(* CoDeSys 2.3.9.47 project: Program-CHP-3.pro *)
(* Libraries: Util.lib 16.5.13 14:00:50, Standard.lib 20.5.14 08:13:26, Iecsfc.lib 16.5.13 14:00:50, SYSLIBCALLBACK.LIB 16.5.13 14:00:50, mod_com.lib 16.5.13 14:00:50, SerComm.lib 16.5.13 14:00:50, Serial_Interface_01.lib 22.4.13 12:50:14, Modb_l05.lib 13.5.15 10:30:08, SysLibTime.lib 16.5.13 14:00:48, SysLibFile.lib 16.5.13 14:00:50, SysLibDir.lib 16.5.13 14:00:50, SysLibMem.lib 16.5.13 14:00:50, WAGO_Datalogger_02.lib 21.4.17 00:23:22, SysLibSockets.lib 22.5.14 16:16:32, NETVARUDP_LIB_V23.LIB 14.6.13 10:36:42 *)

(* PLC configuration (modules and I/O channels)
xDI_24V_01 AT %IX86.0 [BOOLOnX_I] Ch_1 Digital input
xDI_24V_02 AT %IX86.1 [BOOLOnX_I] Ch_2 Digital input
xDI_24V_03 AT %IX86.2 [BOOLOnX_I] Ch_3 Digital input
xDI_24V_04 AT %IX86.3 [BOOLOnX_I] Ch_4 Digital input
xDI_24V_05 AT %IX86.4 [BOOLOnX_I] Ch_5 Digital input
xDI_24V_06 AT %IX86.5 [BOOLOnX_I] Ch_6 Digital input
xDI_24V_07 AT %IX86.6 [BOOLOnX_I] Ch_7 Digital input
xDI_24V_08 AT %IX86.7 [BOOLOnX_I] Ch_8 Digital input
xDO_24V_01 AT %QX24.0 [BOOLOnX_Q] Ch_1 Digital output
xDO_24V_02 AT %QX24.1 [BOOLOnX_Q] Ch_2 Digital output
xDO_24V_03 AT %QX24.2 [BOOLOnX_Q] Ch_3 Digital output
xDO_24V_04 AT %QX24.3 [BOOLOnX_Q] Ch_4 Digital output
xDO_24V_05 AT %QX24.4 [BOOLOnX_Q] Ch_5 Digital output
xDO_24V_06 AT %QX24.5 [BOOLOnX_Q] Ch_6 Digital output
xDO_24V_07 AT %QX24.6 [BOOLOnX_Q] Ch_7 Digital output
xDO_24V_08 AT %QX24.7 [BOOLOnX_Q] Ch_8 Digital output
xDO_24V_09 AT %QX24.8 [BOOLOnX_Q] Ch_1 Digital output
xDO_24V_10 AT %QX24.9 [BOOLOnX_Q] Ch_2 Digital output
xDO_24V_11 AT %QX24.10 [BOOLOnX_Q] Ch_3 Digital output
xDO_24V_12 AT %QX24.11 [BOOLOnX_Q] Ch_4 Digital output
xDO_24V_13 AT %QX24.12 [BOOLOnX_Q] Ch_5 Digital output
xDO_24V_14 AT %QX24.13 [BOOLOnX_Q] Ch_6 Digital output
xDO_24V_15 AT %QX24.14 [BOOLOnX_Q] Ch_7 Digital output
xDO_24V_16 AT %QX24.15 [BOOLOnX_Q] Ch_8 Digital output
AT %IB0 [BYTEOnB_I] First Byte of 24
AT %QB0 [BYTEOnB_Q] First Byte of 24
wAO_U_01 AT %QW12 [WORDOnW_Q] Ch_1 Analog output
wAO_U_02 AT %QW13 [WORDOnW_Q] Ch_2 Analog output
wAO_U_03 AT %QW14 [WORDOnW_Q] Ch_3 Analog output
wAO_U_04 AT %QW15 [WORDOnW_Q] Ch_4 Analog output
wAO_I_01 AT %QW16 [WORDOnW_Q] Ch_1 Analog output
wAO_I_02 AT %QW17 [WORDOnW_Q] Ch_2 Analog output
wAO_I_03 AT %QW18 [WORDOnW_Q] Ch_3 Analog output
wAO_I_04 AT %QW19 [WORDOnW_Q] Ch_4 Analog output
wAO_I_05 AT %QW20 [WORDOnW_Q] Ch_1 Analog output
wAO_I_06 AT %QW21 [WORDOnW_Q] Ch_2 Analog output
wAO_I_07 AT %QW22 [WORDOnW_Q] Ch_3 Analog output
wAO_I_08 AT %QW23 [WORDOnW_Q] Ch_4 Analog output
0750-0459 4 AI 0-10V DC s.e. [Type_8_4_Channels] node 7, in %IB188 out %QB88
  wAI_U_01 AT %IW12 [WORDOnW_I] Ch_1 Input word
  wAI_U_02 AT %IW13 [WORDOnW_I] Ch_2 Input word
  wAI_U_03 AT %IW14 [WORDOnW_I] Ch_3 Input word
  wAI_U_04 AT %IW15 [WORDOnW_I] Ch_4 Input word
0750-0455 4 AI 4-20mA s.e. [Type_8_4_Channels] node 8, in %IB188 out %QB96
  wAI_I_01 AT %IW16 [WORDOnW_I] Ch_1 Input word
  wAI_I_02 AT %IW17 [WORDOnW_I] Ch_2 Input word
  wAI_I_03 AT %IW18 [WORDOnW_I] Ch_3 Input word
  wAI_I_04 AT %IW19 [WORDOnW_I] Ch_4 Input word
  wAI_I_05 AT %IW20 [WORDOnW_I] Ch_1 Input word
  wAI_I_06 AT %IW21 [WORDOnW_I] Ch_2 Input word
  wAI_I_07 AT %IW22 [WORDOnW_I] Ch_3 Input word
  wAI_I_08 AT %IW23 [WORDOnW_I] Ch_4 Input word
0750-0469 2 AI Thermocouple / K / Diag. [Type_44_2_Channels] node 10, in %IB204 out %QB96
  iAI_PTTK_01 AT %IW24 [INTOnW_I] Ch_1 signed Input value
  iAI_PTTK_02 AT %IW25 [INTOnW_I] Ch_2 signed Input value
0750-0469 2 AI Thermocouple / K / Diag. [Type_44_2_Channels] node 11, in %IB212 out %QB96
  iAI_PTTK_03 AT %IW26 [INTOnW_I] Ch_1 signed Input value
  iAI_PTTK_04 AT %IW27 [INTOnW_I] Ch_2 signed Input value
0750-0469 2 AI Thermocouple / K / Diag. [Type_44_2_Channels] node 12, in %IB216 out %QB96
  iAI_PTTK_05 AT %IW28 [INTOnW_I] Ch_1 signed Input value
  iAI_PTTK_06 AT %IW29 [INTOnW_I] Ch_2 signed Input value
0750-0469 2 AI Thermocouple / K / Diag. [Type_44_2_Channels] node 13, in %IB220 out %QB96
  iAI_PTTK_07 AT %IW30 [INTOnW_I] Ch_1 signed Input value
  iAI_PTTK_08 AT %IW31 [INTOnW_I] Ch_2 signed Input value
0750-0469 2 AI Thermocouple / K / Diag. [Type_44_2_Channels] node 14, in %IB224 out %QB96
  iAI_PTTK_09 AT %IW32 [INTOnW_I] Ch_1 signed Input value
  iAI_PTTK_10 AT %IW33 [INTOnW_I] Ch_2 signed Input value
0750-0469 2 AI Thermocouple / K / Diag. [Type_44_2_Channels] node 15, in %IB228 out %QB96
  iAI_PTTK_11 AT %IW34 [INTOnW_I] Ch_1 signed Input value
  iAI_PTTK_12 AT %IW35 [INTOnW_I] Ch_2 signed Input value
0750-0469 2 AI Thermocouple / K / Diag. [Type_44_2_Channels] node 16, in %IB232 out %QB96
  iAI_PTTK_13 AT %IW36 [INTOnW_I] Ch_1 signed Input value
  iAI_PTTK_14 AT %IW37 [INTOnW_I] Ch_2 signed Input value
0750-0469 2 AI Thermocouple / K / Diag. [Type_44_2_Channels] node 17, in %IB236 out %QB96
  iAI_PTTK_15 AT %IW38 [INTOnW_I] Ch_1 signed Input value
  iAI_PTTK_16 AT %IW39 [INTOnW_I] Ch_2 signed Input value
0750-0469 2 AI Thermocouple / K / Diag. [Type_44_2_Channels] node 18, in %IB240 out %QB96
  iAI_PTTK_17 AT %IW40 [INTOnW_I] Ch_1 signed Input value
  iAI_PTTK_18 AT %IW41 [INTOnW_I] Ch_2 signed Input value
0750-0469 2 AI Thermocouple / K / Diag. [Type_44_2_Channels] node 19, in %IB244 out %QB96
  iAI_PTTK_19 AT %IW42 [INTOnW_I] Ch_1 signed Input value
  iAI_PTTK_20 AT %IW43 [INTOnW_I] Ch_2 signed Input value
0750-0469 2 AI Thermocouple / K / Diag. [Type_44_2_Channels] node 20, in %IB248 out %QB96
  iAI_PTTK_21 AT %IW44 [INTOnW_I] Ch_1 signed Input value
  iAI_PTTK_22 AT %IW45 [INTOnW_I] Ch_2 signed Input value
  iAI_PT100_01 AT %IW46 [INTOnW_I] Ch_1 signed Input value
  iAI_PT100_02 AT %IW47 [INTOnW_I] Ch_2 signed Input value
  iAI_PT100_03 AT %IW48 [INTOnW_I] Ch_1 signed Input value
  iAI_PT100_04 AT %IW49 [INTOnW_I] Ch_2 signed Input value
0750-0461 2 AI PT100 (RTD) [Type_44_2_Channels] node 23, in %IB260 out %QB96
  iAI_PT100_05 AT %IW50 [INTOnW_I] Ch_1 signed Input value
  iAI_PT100_06 AT %IW51 [INTOnW_I] Ch_2 signed Input value
0750-0461 2 AI PT100 (RTD) [Type_44_2_Channels] node 24, in %IB264 out %QB96
  iAI_PT100_07 AT %IW52 [INTOnW_I] Ch_1 signed Input value
  iAI_PT100_08 AT %IW53 [INTOnW_I] Ch_2 signed Input value
0750-0461 2 AI PT100 (RTD) [Type_44_2_Channels] node 25, in %IB268 out %QB96
  iAI_PT100_09 AT %IW54 [INTOnW_I] Ch_1 signed Input value
  iAI_PT100_10 AT %IW55 [INTOnW_I] Ch_2 signed Input value
0750-0461 2 AI PT100 (RTD) [Type_44_2_Channels] node 26, in %IB272 out %QB96
  iAI_PT100_11 AT %IW56 [INTOnW_I] Ch_1 signed Input value
  iAI_PT100_12 AT %IW57 [INTOnW_I] Ch_2 signed Input value
0750-0461 2 AI PT100 (RTD) [Type_44_2_Channels] node 27, in %IB276 out %QB96
  iAI_PT100_13 AT %IW58 [INTOnW_I] Ch_1 signed Input value
  iAI_PT100_14 AT %IW59 [INTOnW_I] Ch_2 signed Input value
0750-0461 2 AI PT100 (RTD) [Type_44_2_Channels] node 28, in %IB280 out %QB96
  iAI_PT100_15 AT %IW60 [INTOnW_I] Ch_1 signed Input value
  iAI_PT100_16 AT %IW61 [INTOnW_I] Ch_2 signed Input value
0750-0461 2 AI PT100 (RTD) [Type_44_2_Channels] node 29, in %IB284 out %QB96
  iAI_PT100_17 AT %IW62 [INTOnW_I] Ch_1 signed Input value
  iAI_PT100_18 AT %IW63 [INTOnW_I] Ch_2 signed Input value
0750-0461 2 AI PT100 (RTD) [Type_44_2_Channels] node 30, in %IB288 out %QB96
  iAI_PT100_19 AT %IW64 [INTOnW_I] Ch_1 signed Input value
  iAI_PT100_20 AT %IW65 [INTOnW_I] Ch_2 signed Input value
0750-0461 2 AI PT100 (RTD) [Type_44_2_Channels] node 31, in %IB292 out %QB96
  iAI_PT100_21 AT %IW66 [INTOnW_I] Ch_1 signed Input value
  iAI_PT100_22 AT %IW67 [INTOnW_I] Ch_2 signed Input value
0750-0461 2 AI PT100 (RTD) [Type_44_2_Channels] node 0, in %IB296 out %QB96
  iAI_PT100_23 AT %IW68 [INTOnW_I] Ch_1 signed Input value
  iAI_PT100_24 AT %IW69 [INTOnW_I] Ch_2 signed Input value
0750-0460 4 AI PT100 (RTD) [Type_44_4_Channels] node 32, in %IB300 out %QB96
  AT %IW70 [INTOnW_I] Ch_1 signed Input value
  AT %IW71 [INTOnW_I] Ch_2 signed Input value
  AT %IW72 [INTOnW_I] Ch_3 signed Input value
  AT %IW73 [INTOnW_I] Ch_4 signed Input value
0750-0460 4 AI PT100 (RTD) [Type_44_4_Channels] node 33, in %IB304 out %QB96
  AT %IW74 [INTOnW_I] Ch_1 signed Input value
  AT %IW75 [INTOnW_I] Ch_2 signed Input value
  AT %IW76 [INTOnW_I] Ch_3 signed Input value
  AT %IW77 [INTOnW_I] Ch_4 signed Input value
0750-0460 4 AI PT100 (RTD) [Type_44_4_Channels] node 34, in %IB312 out %QB96
  AT %IW78 [INTOnW_I] Ch_1 signed Input value
  AT %IW79 [INTOnW_I] Ch_2 signed Input value
  AT %IW80 [INTOnW_I] Ch_3 signed Input value
  AT %IW81 [INTOnW_I] Ch_4 signed Input value
0750-0460 4 AI PT100 (RTD) [Type_44_4_Channels] node 35, in %IB320 out %QB96
  AT %IW82 [INTOnW_I] Ch_1 signed Input value
  AT %IW83 [INTOnW_I] Ch_2 signed Input value
  AT %IW84 [INTOnW_I] Ch_3 signed Input value
  AT %IW85 [INTOnW_I] Ch_4 signed Input value
Modbus variables [PFC200MODBUS] node 1, in %IB0 out %QB0 {PlcStopBehaviour = 1; FiledbusErrorBehaviour = 1; TcpOperation = 1; TcpPort = 502; TcpTimeout = 600; UdpOperation = 1; UdpPort = 502; RtuOperation = 0; NodeId = 1; ResponseTimeout = 5000; Interface = 0; Baud = 115200; StopBits = 1; Parity = 1; FlowCtrl = 0; PhysInterface = 0}
Modbus-Master [MB_MASTER] node 2, in %IB0 out %QB0
*)

(* Task configuration *)
TASK PLC_PRG (PRIORITY := 14, INTERVAL := T#200ms);
	PLC_PRG();
END_TASK

(* Global variable list: Constant_Values *)
VAR_GLOBAL
	oil_specific_heat_0: REAL := 2.1415;
	oil_specific_heat_20: REAL := 2.1541;
	oil_specific_heat_40: REAL := 2.1667;
	oil_specific_heat_60: REAL := 2.1792;
	oil_specific_heat_80: REAL := 2.1918;
	oil_specific_heat_100: REAL := 2.2044;
	oil_specific_heat_120: REAL := 2.2169;
	oil_specific_heat_140: REAL := 2.2295;
	oil_specific_heat_160: REAL := 2.2420;
	oil_specific_heat_180: REAL := 2.2546;
	oil_specific_heat_200: REAL := 2.2672;
	oil_specific_heat_220: REAL := 2.2797;
	oil_specific_heat_240: REAL := 2.2923;
	oil_specific_heat_260: REAL := 2.3048;

	oil_density_0: REAL := 906;
	oil_density_20: REAL := 895;
	oil_density_40: REAL := 883;
	oil_density_60: REAL := 874;
	oil_density_80: REAL := 862;
	oil_density_100: REAL := 850;
	oil_density_120: REAL := 838;
	oil_density_140: REAL := 825;
	oil_density_160: REAL := 813;
	oil_density_180: REAL := 800;
	oil_density_200: REAL := 788;
	oil_density_220: REAL := 775;
	oil_density_240: REAL := 760;
	oil_density_260: REAL := 747;

	(* shutdown parameters *)
	oil_shutdown_temp: REAL := 210;
	water_shutdown_temp: REAL := 210;
	flue_shutdown_temp: REAL := 300;

END_VAR

(* Global variable list: Global_Variables *)
VAR_GLOBAL

(*Flue gas parameters*)
	
	flue_gas_temp_01: REAL;
	flue_gas_temp_02: REAL;
	flue_gas_temp_03: REAL;
	flue_gas_temp_04: REAL;
	flue_gas_temp_05: REAL;
	flue_gas_temp_06: REAL;
	
(*Oil temperature, pressure and flow*)
	
	oil_temp_01: REAL;
	oil_temp_02: REAL;
	oil_temp_03: REAL;
	oil_temp_04: REAL;
	oil_temp_05: REAL;
	oil_temp_06: REAL;
	oil_temp_07: REAL;
	oil_temp_08: REAL;
	oil_temp_09: REAL;
	oil_temp_10: REAL;

	oil_pump_01_start: BOOL;   (* Start/Stop oil pump*)
	oil_pump_01_set: REAL;   (*Speed regulation of the oil pump*)
	oil_pump_01_value: REAL;   (*Speed of the oil pump (inverter response)*)
	oil_pump_01_status: BOOL;   (*Status of the oil pump operation*)
	
	oil_flow_01_start: BOOL;   (* Start/stop oil flowmeter no. 1*)
	oil_flow_01_value: REAL;   (* Measured oil flow (dm3/MIN) - flowmeter no. 1*)
	oil_flow_02_start: BOOL;  (*Start/stop oil flowmeter no. 2*)
	oil_flow_02_value: REAL;   (* Measured oil flow (dm3/min) - flowmeter no. 2*)

(*Water temperature, pressure and flow*)
		
	water_temp_01: REAL;
	water_temp_02: REAL;
	water_temp_03: REAL;
	water_temp_04: REAL;
	water_temp_05: REAL;
	water_temp_06: REAL;
	water_temp_07: REAL;
	water_temp_08: REAL;
	water_temp_09: REAL;
	water_temp_10: REAL;
	water_temp_11: REAL;
	water_temp_12: REAL;

	water_pump_01_power: BOOL;  (* Power on/off of the water pump no. 1*)
	water_pump_01_start: BOOL;   (* Start/Stop water pump no. 1*)
	water_pump_01_set: REAL;   (* Speed regulation of the water pump no. 1*)
	water_pump_02_power: BOOL;  (* Power on/off of the water pump no. 2*)
	water_pump_02_start: BOOL;   (* Start/Stop water pump no. 2*)
	water_pump_02_set: REAL;   (* Speed regulation of the water pump no. 2*)
	
	water_flow_01_start: BOOL;   (*Start/stop water flowmeter *)
	water_flow_01_value: REAL;   (* Measured water flow (m3/h) - water flowmeter no. 1*)

(*Fans and pumps control*)
	
	air_fan_01_start: BOOL;   (* Start/Stop inlet air fan*)
	air_fan_01_set: REAL;   (* Speed regulation of the inlet air fan*)
	air_fan_01_value: REAL;   (* Speed of the inlet air fan (inverter response)*)
	air_fan_01_status: BOOL;   (*Status OF the inlet air fan operation*)

	air_fan_02_start: BOOL;   (* Start/Stop outlet air fan*)
	air_fan_02_set: REAL;   (* Speed regulation of the outlet air fan*)
	air_fan_02_value: REAL;   (*Speed of the outlet air fan (inverter response)*)
	air_fan_02_status: BOOL;   (* Status OF the outlet air fan operation*)

	air_fan_03_start_fwd: BOOL;
	air_fan_03_start_rwd: BOOL;
	air_fan_03_set: REAL;
	air_fan_03_value: REAL;

(*Condensate level*)
	condensate_level_01_start: BOOL;
	condensate_level_01_value: REAL;

(*Steam pressure*)
	steam_pressure_01_start: BOOL;
	steam_pressure_01_value: REAL;

	INIT: BOOL := TRUE;
	AUXILIARY_EXCHANGER_ON : BOOL := FALSE;

END_VAR

(* Global variable list: Networkmanagement implicit Variables UDP *)
VAR_GLOBAL CONSTANT
	USE_NWVARS_UDP : BOOL := FALSE;
	MAX_NetVarItems_UDP	: INT := 0;
	MAX_NetVarPDO_Rx_UDP	: INT := 0;
	MAX_NetVarPDO_Tx_UDP	: INT := 0;
	MAX_NetVarOD_UDP		: INT := 0;
END_VAR
VAR_GLOBAL
	pNetVarItems_UDP		: ARRAY[0..MAX_NetVarItems_UDP] OF NetVarDataItem_UDP;
	pNetVarPDO_Rx_UDP		: ARRAY[0..MAX_NetVarPDO_Rx_UDP] OF NetVarPDO_Rx_UDP;
	pNetVarPDO_Tx_UDP		: ARRAY[0..MAX_NetVarPDO_Tx_UDP] OF NetVarPDO_Tx_UDP;
	pNetVarOD_UDP			: ARRAY[0..MAX_NetVarOD_UDP] OF NetVarSDO_UDP;
	pNetVarPDO_Rx_Diagnosis_UDP : ARRAY[0..MAX_NetVarPDO_Rx_UDP] OF NetVarUDPDiagStruct;
	pNetVarPDO_Tx_Diagnosis_UDP : ARRAY[0..MAX_NetVarPDO_Tx_UDP] OF NetVarUDPDiagStruct;
END_VAR

(* POU PLC_PRG, ST *)
PROGRAM PLC_PRG
VAR
	Boiler_Power: OIL_POWER;
	Oil_Water_Heat_Exchanger_Oil_Side_Power: OIL_POWER;
	Oil_Water_Heat_Exchanger_Water_Side_Power: WATER_POWER;
	Tank_Power: WATER_POWER;
	Control_Program: BOILER_PROGRAM;
END_VAR
(* Read all inputs *)

(*Inlet air fan operation parameters*)
	air_fan_01_value		:=		WORD_TO_REAL(wAI_I_01) / 327.67;   					(*Response from inverter*)
	air_fan_01_status	:=		xDI_24V_01;  												(*Status of the inlet air fan operation*)

(*Flue gas fan operation parameters*)
	air_fan_02_value		:=		WORD_TO_REAL(wAI_I_02) / 327.67;  					(*Response from inverter*)
	air_fan_02_status	:=		xDI_24V_02;  												(*Status of the outlet air fan operation*)

(*Flue gas temperature conversion*)
	flue_gas_temp_01	:= 		INT_TO_REAL(iAI_PT100_23)/10;  						(*Pt100 sensor located in the inlet to chimney*)
	flue_gas_temp_02	:= 		INT_TO_REAL(iAI_PTTK_01)/10;							(*PTTK sensor (4p) located in the second combustion chamber*)
	flue_gas_temp_03	:= 		INT_TO_REAL(iAI_PTTK_02)/10;  						(*PTTK sensor (4p) located in the second combustion chamber*)
	flue_gas_temp_04	:= 		INT_TO_REAL(iAI_PTTK_03)/10;   						(*PTTK sensor (4p) located in the second combustion chamber*)
	flue_gas_temp_05	:= 		INT_TO_REAL(iAI_PTTK_04)/10;  						(*PTTK sensor (4p) located in the second combustion chamber*)
	flue_gas_temp_06	:= 		INT_TO_REAL(iAI_PTTK_05)/10;   						(*PTTK sensor located in the first combustion chamber*)

(*Oil temperature measurements*)
	oil_temp_01			:= 		INT_TO_REAL(iAI_PT100_01)/10;  						(*Pt100 sensor no. 1*)
	oil_temp_02			:=		INT_TO_REAL(iAI_PT100_02)/10;  						(*Pt100 sensor no. 2*)
	oil_temp_03 			:= 		INT_TO_REAL(iAI_PT100_03)/10;  						(*Pt100 sensor no. 3*)
	oil_temp_04 			:=		INT_TO_REAL(iAI_PT100_04)/10;   						(*Pt100 sensor no. 4*)
	oil_temp_05 			:=		INT_TO_REAL(iAI_PT100_05)/10;   						(*Pt100 sensor no. 5*)
	oil_temp_06			:=		INT_TO_REAL(iAI_PT100_06)/10;   						(*Pt100 sensor no. 6*)
	oil_temp_07			:= 		INT_TO_REAL(iAI_PT100_07)/10;  						(*Pt100 sensor no. 7*)
	oil_temp_08			:=		INT_TO_REAL(iAI_PT100_08)/10;   						(*Pt100 sensor no. 8*)
	oil_temp_09			:=		INT_TO_REAL(iAI_PT100_09)/10;  						(*Pt100 sensor no. 9*)
	oil_temp_10			:= 		INT_TO_REAL(iAI_PT100_10)/10;   						(*Pt100 sensor no. 10*)

(*Oil pump parameters*)
	oil_pump_01_value 	:= 		WORD_TO_REAL(wAI_I_03) / 327.67;   					(*Response from inverter*)
	oil_pump_01_status	:= 		xDI_24V_03;   												(*Status of the oil pump operation*)

(*Oil flowmeters parameters*)
	oil_flow_01_value 	:= 		WORD_TO_REAL(wAI_I_04) / 327.67;    					(*flow in dm3/min, max. 100 dm3/min *)

	oil_flow_02_value 	:= 		WORD_TO_REAL(wAI_I_05) / 327.67;    					(*flow in dm3/min, max. 100 dm3/min*)
	
(*Water temperature measurements*)
	water_temp_01 		:= 		INT_TO_REAL(iAI_PT100_11)/10;   						(*Pt100 sensor no. 11*)
	water_temp_02 		:= 		INT_TO_REAL(iAI_PT100_12)/10;  						(*Pt100 sensor no. 12*)
	water_temp_03 		:= 		INT_TO_REAL(iAI_PT100_13)/10;  						(*Pt100 sensor no. 13*)
	water_temp_04 		:= 		INT_TO_REAL(iAI_PT100_14)/10;   						(*Pt100 sensor no. 14*)
	water_temp_05 		:= 		INT_TO_REAL(iAI_PT100_15)/10;   						(*Pt100 sensor no. 15*)
	water_temp_06 		:= 		INT_TO_REAL(iAI_PT100_16)/10;   						(*Pt100 sensor no. 16*)
	water_temp_07 		:= 		INT_TO_REAL(iAI_PT100_17)/10;   						(*Pt100 sensor no. 17*)
	water_temp_08 		:= 		INT_TO_REAL(iAI_PT100_18)/10;   						(*Pt100 sensor no. 18*)
	water_temp_09 		:= 		INT_TO_REAL(iAI_PT100_19)/10;   						(*Pt100 sensor no. 19*)
	water_temp_10 		:= 		INT_TO_REAL(iAI_PT100_20)/10;   						(*Pt100 sensor no. 20*)
	water_temp_11		:=		INT_TO_REAL(iAI_PT100_21)/10;						(*Pt100 sensor no. 21*)
	water_temp_12		:=		INT_TO_REAL(iAI_PT100_22)/10;						(*Pt100 sensor no. 22*)

(*Water flowmeter parameters*)
	water_flow_01_value 	:= 		WORD_TO_REAL(wAI_I_06) / 5461.2;   					(*flow in m3/h, max. 6 m3/h*)

(*Water cooler air fan*)
	air_fan_03_value		:=		WORD_TO_REAL(wAI_U_01) / 327.67;

(*Power of the boiler*)
Boiler_Power(
	oil_flow				:=		oil_flow_01_value,
	oil_temp_low			:=		oil_temp_02,
	oil_temp_high			:=		oil_temp_01,
	oil_temp_conv		:=		oil_temp_02,
	OIL_POWER=> );

(*Power transferred from oil to water in oil-water heat exchanger*)
Oil_Water_Heat_Exchanger_Oil_Side_Power(
	oil_flow				:=		oil_flow_01_value,
	oil_temp_low			:=		oil_temp_06,
	oil_temp_high			:=		oil_temp_05,
	oil_temp_conv		:=		oil_temp_02,
	OIL_POWER=> );

(*Power received by water tank*)
	Tank_Power(
	water_flow:= water_flow_01_value,
	water_temp_high:= water_temp_04,
	water_temp_low:= water_temp_03,
	WATER_POWER=> );


(*Power received by water from oil in oil-water heat exchanger*)
	Oil_Water_Heat_Exchanger_Water_Side_Power(
	water_flow:= water_flow_01_value,
	water_temp_high:= water_temp_01,
	water_temp_low:= water_temp_02,
	WATER_POWER=> );

(*Condensate level*)
	condensate_level_01_value		:=		WORD_TO_REAL(wAI_I_08) / 23.57;    					(*Condensate level in mm*)

(*Steam pressure*)
	steam_pressure_01_value		:=		WORD_TO_REAL(wAI_I_07) / 2047.94; 					(*pressure in bars*)


(* Controll program *)

	Control_Program();

(* Write to all outputs *)

(*Inlet air fan operation parameters*)
	xDO_24V_01			:=		air_fan_01_start;  											(*Start/stop inlet air fan*)
	IF air_fan_01_set <= 30 THEN
		wAO_U_01		:=		0;  															(*Set value of the inlet air fan*)
	ELSE
		wAO_U_01		:=		REAL_TO_WORD(((air_fan_01_set  - 30) * 1.42857) * 327.67);
	END_IF;
	IF wAO_U_01 >32767 THEN
		wAO_U_01		:= 		32767;
	END_IF;

(*Flue gas fan operation parameters*)
	xDO_24V_02			:=		air_fan_02_start;  											(*Start/stop outlet air fan*)
	wAO_U_02			:= 		REAL_TO_WORD(air_fan_02_set * 327.67);   			(*Set value of the outlet air fan*)

(*Oil pump parameters*)
	xDO_24V_03 			:= 		oil_pump_01_start;   										(*Start/stop oil pump*)
	wAO_U_03			:= 		REAL_TO_WORD(oil_pump_01_set * 327.67);  		(*Set value of the pump speed*)

(*Oil flowmeters parameters*)
	xDO_24V_11 			:= 		oil_flow_01_start;   										(*Turn on/turn off oil flowmeter no. 1*)

	xDO_24V_12 			:= 		oil_flow_02_start;   										(*Turn on/turn off oil flowmeter no. 2*)

(*Water pumps parameters*)
	xDO_24V_04			:= 		water_pump_01_power;  								(*Turn on/turn off water pump no. 1*)
	xDO_24V_05 			:= 		water_pump_01_start;   									(*Start/stop water pump no. 1*)
	wAO_I_01 				:= 		REAL_TO_WORD(water_pump_01_set * 327.67);   	(*Set value of the water pump no. 1 speed*)

	xDO_24V_06 			:= 		water_pump_02_power;   								(*Turn on/turn off water pump no. 2*)
	xDO_24V_07 			:= 		water_pump_02_start;   									(*Start/stop water pump no. 2*)
	wAO_I_02 				:= 		REAL_TO_WORD(water_pump_02_set * 327.67);   	(*Set value of the water pump no. 2 speed*)

(*Water flowmeter parameters*)
	xDO_24V_13 			:= 		water_flow_01_start;   									(*Turn on/turn off water flowmeter *)

(*Water cooler air fan*)
	xDO_24V_09			:=		air_fan_03_start_fwd;
	xDO_24V_10			:=		air_fan_03_start_rwd;
	wAO_I_03				:=		REAL_TO_WORD(air_fan_03_set*327.67);

(*Condensate level*)
	xDO_24V_16						:=		condensate_level_01_start;								(*Turn on/turn off condensate  level meter *)

(*Steam pressure*)
	xDO_24V_15						:=		steam_pressure_01_start;								(*Turn on/turn off pressure  *)
END_PROGRAM

(* POU OIL_POWER, ST *)
FUNCTION_BLOCK OIL_POWER
VAR_INPUT
	oil_flow:				REAL;			(*oil flow in l/min*)
	oil_temp_low:			REAL;			(*cold oil temperature at the inlet to the boiler*)
	oil_temp_high:		REAL;			(*hot oil temperature at the outlet from the boiler*)
	oil_temp_conv:		REAL;			(*oil temperature to specific heat and density conversion - temperature measured close to the flowmeter*)
END_VAR
VAR
	oil_specific_heat: 		REAL;
	oil_density: 			REAL;
END_VAR
VAR_OUTPUT
	OIL_POWER:			REAL;
END_VAR
(* Oil specific heat*)

IF oil_temp_conv >= 0 AND oil_temp_conv <20 THEN
	oil_specific_heat := oil_specific_heat_0 + ((oil_temp_conv / 20) * (oil_specific_heat_20 - oil_specific_heat_0));
ELSIF oil_temp_conv >= 20 AND oil_temp_conv <40 THEN
	oil_specific_heat := oil_specific_heat_20 + (((oil_temp_conv - 20) / 20) * (oil_specific_heat_40 - oil_specific_heat_20));
ELSIF oil_temp_conv >= 40 AND oil_temp_conv <60 THEN
	oil_specific_heat := oil_specific_heat_40 + (((oil_temp_conv - 40) / 20) * (oil_specific_heat_60 - oil_specific_heat_40));
ELSIF oil_temp_conv >= 60 AND oil_temp_conv <80 THEN
	oil_specific_heat := oil_specific_heat_60 + (((oil_temp_conv - 60) / 20) * (oil_specific_heat_80 - oil_specific_heat_60));
ELSIF oil_temp_conv >= 80 AND oil_temp_conv <100 THEN
	oil_specific_heat := oil_specific_heat_80 + (((oil_temp_conv - 80) / 20) * (oil_specific_heat_100 - oil_specific_heat_80));
ELSIF oil_temp_conv >= 100 AND oil_temp_conv <120 THEN
	oil_specific_heat := oil_specific_heat_100 + (((oil_temp_conv - 100) / 20) * (oil_specific_heat_120 - oil_specific_heat_100));
ELSIF oil_temp_conv >= 120 AND oil_temp_conv <140 THEN
	oil_specific_heat := oil_specific_heat_120 + (((oil_temp_conv - 120) / 20) * (oil_specific_heat_140 - oil_specific_heat_120));
ELSIF oil_temp_conv >= 140 AND oil_temp_conv <160 THEN
	oil_specific_heat := oil_specific_heat_140 + (((oil_temp_conv - 140) / 20) * (oil_specific_heat_160 - oil_specific_heat_140));
ELSIF oil_temp_conv >= 160 AND oil_temp_conv <180 THEN
	oil_specific_heat := oil_specific_heat_160 + (((oil_temp_conv - 160) / 20) * (oil_specific_heat_180 - oil_specific_heat_160));
ELSIF oil_temp_conv >= 180 AND oil_temp_conv <200 THEN
	oil_specific_heat := oil_specific_heat_180 + (((oil_temp_conv - 180) / 20) * (oil_specific_heat_200 - oil_specific_heat_180));
ELSIF oil_temp_conv >= 200 AND oil_temp_conv <220 THEN
	oil_specific_heat := oil_specific_heat_200 + (((oil_temp_conv - 200) / 20) * (oil_specific_heat_220 - oil_specific_heat_200));
ELSIF oil_temp_conv >= 220 AND oil_temp_conv <240 THEN
	oil_specific_heat := oil_specific_heat_220 + (((oil_temp_conv - 220) / 20) * (oil_specific_heat_240 - oil_specific_heat_220));
ELSIF oil_temp_conv >= 240 AND oil_temp_conv <260 THEN
	oil_specific_heat := oil_specific_heat_240 + (((oil_temp_conv - 240) / 20) * (oil_specific_heat_260 - oil_specific_heat_240));
END_IF

(*Oil density*)

IF oil_temp_conv >= 0 AND oil_temp_conv <20 THEN
	oil_density := oil_density_0 + ((oil_temp_conv / 20) * (oil_density_20 - oil_density_0));
ELSIF oil_temp_conv >= 20 AND oil_temp_conv <40 THEN
	oil_density := oil_density_20 + (((oil_temp_conv - 20) / 20) * (oil_density_40 - oil_density_20));
ELSIF oil_temp_conv >= 40 AND oil_temp_conv <60 THEN
	oil_density := oil_density_40 + (((oil_temp_conv - 40) / 20) * (oil_density_60 - oil_density_40));
ELSIF oil_temp_conv >= 60 AND oil_temp_conv <80 THEN
	oil_density := oil_density_60 + (((oil_temp_conv - 60) / 20) * (oil_density_80 - oil_density_60));
ELSIF oil_temp_conv >= 80 AND oil_temp_conv <100 THEN
	oil_density := oil_density_80 + (((oil_temp_conv - 80) / 20) * (oil_density_100 - oil_density_80));
ELSIF oil_temp_conv >= 100 AND oil_temp_conv <120 THEN
	oil_density := oil_density_100 + (((oil_temp_conv - 100) / 20) * (oil_density_120 - oil_density_100));
ELSIF oil_temp_conv >= 120 AND oil_temp_conv <140 THEN
	oil_density := oil_density_120 + (((oil_temp_conv - 120) / 20) * (oil_density_140 - oil_density_120));
ELSIF oil_temp_conv >= 140 AND oil_temp_conv <160 THEN
	oil_density := oil_density_140 + (((oil_temp_conv - 140) / 20) * (oil_density_160 - oil_density_140));
ELSIF oil_temp_conv >= 160 AND oil_temp_conv <180 THEN
	oil_density := oil_density_160 + (((oil_temp_conv - 160) / 20) * (oil_density_180 - oil_density_160));
ELSIF oil_temp_conv >= 180 AND oil_temp_conv <200 THEN
	oil_density := oil_density_180 + (((oil_temp_conv - 180) / 20) * (oil_density_200 - oil_density_180));
ELSIF oil_temp_conv >= 200 AND oil_temp_conv <220 THEN
	oil_density := oil_density_200 + (((oil_temp_conv - 200) / 20) * (oil_density_220 - oil_density_200));
ELSIF oil_temp_conv >= 220 AND oil_temp_conv <240 THEN
	oil_density := oil_density_220 + (((oil_temp_conv - 220) / 20) * (oil_density_240 - oil_density_220));
ELSIF oil_temp_conv >= 240 AND oil_temp_conv <260 THEN
	oil_density := oil_density_240 + (((oil_temp_conv - 240) / 20) * (oil_density_260 - oil_density_240));
END_IF

oil_power := (oil_flow * oil_density / 60000) * oil_specific_heat * (oil_temp_high - oil_temp_low);					(*power in kJ/s = kW*)
END_FUNCTION_BLOCK

(* POU WATER_POWER, ST *)
FUNCTION_BLOCK WATER_POWER
VAR_INPUT
	water_flow: REAL;
	water_temp_high: REAL;
	water_temp_low: REAL;
END_VAR
VAR_OUTPUT
	WATER_POWER: REAL;
END_VAR
VAR
	water_specific_heat: REAL := 4.19;
END_VAR
water_power := (water_flow  / 3.6) * water_specific_heat * (water_temp_high - water_temp_low);					(*power in kJ/s = kW*)
END_FUNCTION_BLOCK

(* POU BOILER_PROGRAM, ST *)
FUNCTION_BLOCK BOILER_PROGRAM
VAR_INPUT
END_VAR
VAR_OUTPUT
END_VAR
VAR
	Flue_Control : FLUE_GAS_CONTROL;
	OIL_CONTROL: OIL_CONTROL;
	WATER_CONTROL : WATER_CONTROL;
END_VAR
(* check if initialization *)

IF INIT THEN
	(* start inlet airfan *)
	air_fan_01_start := TRUE;
	air_fan_01_set := 50;

	(* start outlet airfan *)
	air_fan_02_start := TRUE;
	air_fan_02_set := 60;

	(* start oil pump *)
	oil_pump_01_start := TRUE;
	oil_pump_01_set := 70;

	(* start water pump *)
	water_pump_01_start := TRUE;
	water_pump_01_set := 70;

	INIT := FALSE;
END_IF

(* control the oil circulation *)

OIL_CONTROL(oil_temp := oil_temp_01, flue_gas_temp := flue_gas_temp_01);

(* control the flue gas circulation *)

Flue_Control(flue_gas_temp := flue_gas_temp_01);

(* control the waterl circulation *)

WATER_CONTROL(water_temp := water_temp_02, water_avg := (water_temp_03 + water_temp_04) / 2);

(* check for emergency shutdown *)

IF water_temp_01 > 95 OR flue_gas_temp_01 > 300 OR oil_temp_01 > 210 THEN

	(* set airfan to minimum *)
	air_fan_01_set := 30;
	air_fan_02_set := 30;

	(* set all pumps to maximum *)
	water_pump_01_set := 100;

	water_pump_02_start := TRUE;
	water_pump_02_set := 100;

	oil_pump_01_set := 100;

	air_fan_03_start_fwd := TRUE;
	air_fan_03_start_rwd := TRUE;
	air_fan_03_set := 100;

	(* set auxiliary exchanger on *)

	AUXILIARY_EXCHANGER_ON := TRUE;
END_IF
END_FUNCTION_BLOCK

(* POU FLUE_GAS_CONTROL, ST *)
FUNCTION_BLOCK FLUE_GAS_CONTROL
VAR_INPUT
	flue_gas_temp: REAL;
END_VAR
VAR_OUTPUT
END_VAR
VAR
	Flue_Timer_01: TON;
	Flue_Timer_02: TON;
	Flue_Timer_03: TON;
	Flue_Timer_04: TON;
	Flue_Timer_05: TON;
	Flue_Timer_06: TON;
END_VAR
Flue_Timer_01(IN := flue_gas_temp < 220, PT := T#30s);

IF Flue_Timer_01.Q THEN
	air_fan_01_set := 60;
	air_fan_02_set := 70;
END_IF

Flue_Timer_02(IN := flue_gas_temp < 200, PT := T#30s);

IF Flue_Timer_02.Q THEN
	air_fan_01_set := 70;
	air_fan_02_set := 80;
END_IF

Flue_Timer_03(IN := flue_gas_temp < 180, PT := T#30s);

IF Flue_Timer_03.Q THEN
	air_fan_01_set := 80;
	air_fan_02_set := 90;
END_IF


Flue_Timer_04(IN := flue_gas_temp > 250, PT := T#30s);

IF Flue_Timer_04.Q THEN
	air_fan_01_set := 40;
	air_fan_02_set := 50;
END_IF

Flue_Timer_05(IN := flue_gas_temp > 265, PT := T#30s);

IF Flue_Timer_05.Q THEN
	air_fan_01_set := 30;
	air_fan_02_set := 40;
END_IF

Flue_Timer_06(IN := flue_gas_temp > 280, PT := T#30s);

IF Flue_Timer_06.Q THEN
	air_fan_01_set := 20;
	air_fan_02_set := 30;
END_IF
END_FUNCTION_BLOCK

(* POU OIL_CONTROL, ST *)
FUNCTION_BLOCK OIL_CONTROL
VAR_INPUT
	oil_temp : REAL;
	flue_gas_temp: REAL;
END_VAR
VAR_OUTPUT
END_VAR
VAR
	Oil_Timer_01: TON;
	Oil_Timer_02: TON;
	Oil_Timer_03: TON;
	Oil_Timer_04: TON;
	Oil_Timer_05: TON;
	Oil_Timer_06: TON;
END_VAR
Oil_Timer_01(IN := oil_temp < 170, PT := T#30s);

IF Oil_Timer_01.Q THEN
	water_pump_01_set := 55;
END_IF

Oil_Timer_02(IN := oil_temp < 155, PT := T#30s);

IF Oil_Timer_02.Q THEN
	water_pump_01_set := 40;
	oil_pump_01_set := 55;
END_IF

Oil_Timer_03(IN := oil_temp < 130, PT := T#30s);

IF Oil_Timer_03.Q THEN
	water_pump_01_set := 30;
	oil_pump_01_set := 40;
END_IF


Oil_Timer_04(IN := oil_temp > 185, PT := T#30s);

IF Oil_Timer_04.Q THEN
	water_pump_01_set := 80;
END_IF

Oil_Timer_05(IN := oil_temp > 195, PT := T#30s);

IF Oil_Timer_05.Q THEN
	water_pump_01_set := 90;
	oil_pump_01_set := 80;
END_IF

Oil_Timer_06(IN := oil_temp > 200, PT := T#30s);

IF Oil_Timer_06.Q THEN
	water_pump_01_set := 100;
	oil_pump_01_set := 90;
END_IF

IF flue_gas_temp < 235 AND (Oil_Timer_01.Q OR Oil_Timer_02.Q OR Oil_Timer_03.Q) THEN
	air_fan_01_set := 60;
	air_fan_02_set := 70;
ELSIF flue_gas_temp > 235 AND (Oil_Timer_04.Q OR Oil_Timer_05.Q OR Oil_Timer_06.Q) THEN
	air_fan_01_set := 40;
	air_fan_02_set := 60;
END_IF
END_FUNCTION_BLOCK

(* POU WATER_CONTROL, ST *)
FUNCTION_BLOCK WATER_CONTROL
VAR_INPUT
	water_temp: REAL;
	water_avg : REAL;
END_VAR
VAR_OUTPUT
END_VAR
VAR
	Water_Timer_01: TON;
	Water_Timer_02: TON;
END_VAR
Water_Timer_01(IN := water_temp > 70, PT := T#30s);

Water_Timer_02(IN := water_temp > 85, PT := T#30s);

IF Water_Timer_01.Q OR water_avg > 50 THEN

	water_pump_02_start := TRUE;
	water_pump_02_set := 70;

	air_fan_03_start_fwd := TRUE;
	air_fan_03_start_rwd := TRUE;
	air_fan_03_set := 50;

	IF Water_Timer_02.Q THEN
		AUXILIARY_EXCHANGER_ON := TRUE;
	ELSE
		AUXILIARY_EXCHANGER_ON := FALSE;
	END_IF

ELSE

	water_pump_02_start := FALSE;
	water_pump_02_set := 0;

	air_fan_03_start_fwd := FALSE;
	air_fan_03_start_rwd := FALSE;
	air_fan_03_set := 0;

	AUXILIARY_EXCHANGER_ON := FALSE;

END_IF
END_FUNCTION_BLOCK

(* POU SAVE_DATA, CFC *)
PROGRAM SAVE_DATA
VAR
	Datalogger_01: FbDatalogger;
	xStart: BOOL;
	xTrigger: BOOL;
	bDtype: BYTE := 1;
	xFirstCycle: BOOL := TRUE;
	i: INT;
END_VAR

VAR RETAIN PERSISTENT
	channels: ARRAY[1.. gc_bMAXCHANNELS] OF typUserInput;
	settings: typConfigDatalogger;
END_VAR
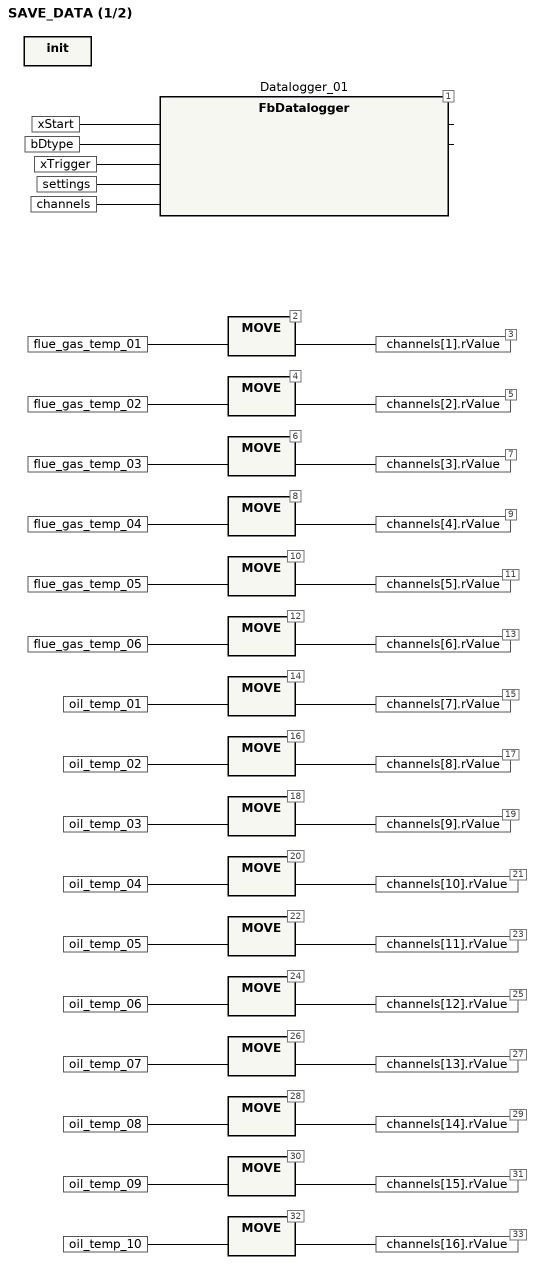
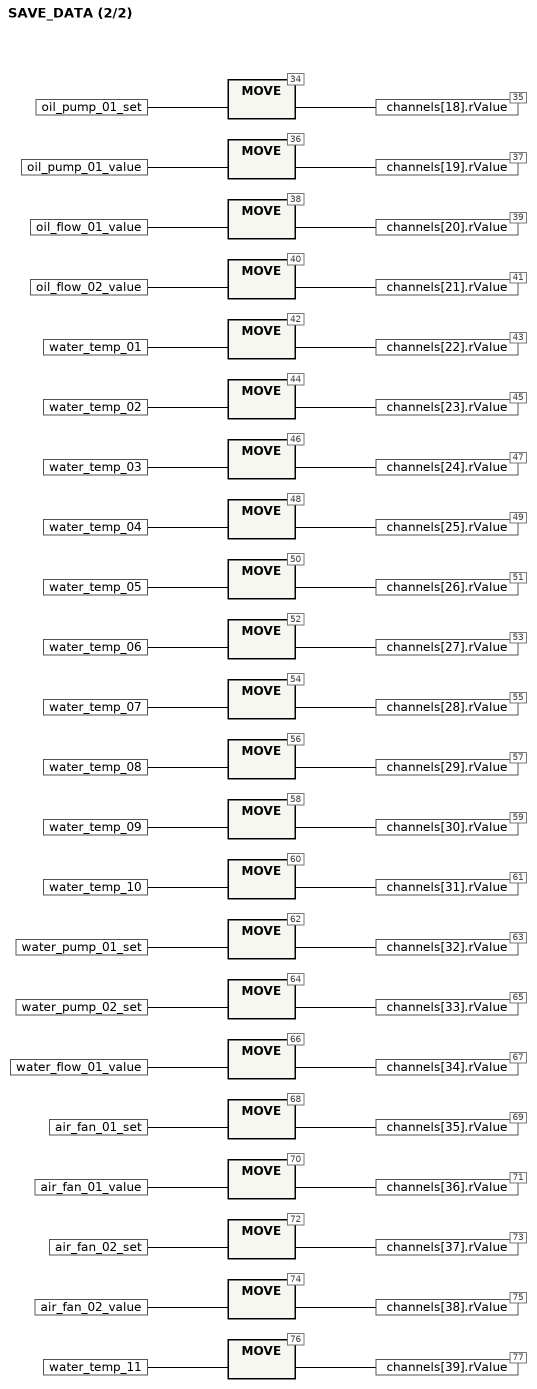
_CFC_ (* Continuous Function Chart, elements in execution order *)
#0 init()
#1 Datalogger_01:FbDatalogger(xStart, bDtype, xTrigger, settings, channels)
#2 MOVE(flue_gas_temp_01)
#3 channels[1].rValue <= #2
#4 MOVE(flue_gas_temp_02)
#5 channels[2].rValue <= #4
#6 MOVE(flue_gas_temp_03)
#7 channels[3].rValue <= #6
#8 MOVE(flue_gas_temp_04)
#9 channels[4].rValue <= #8
#10 MOVE(flue_gas_temp_05)
#11 channels[5].rValue <= #10
#12 MOVE(flue_gas_temp_06)
#13 channels[6].rValue <= #12
#14 MOVE(oil_temp_01)
#15 channels[7].rValue <= #14
#16 MOVE(oil_temp_02)
#17 channels[8].rValue <= #16
#18 MOVE(oil_temp_03)
#19 channels[9].rValue <= #18
#20 MOVE(oil_temp_04)
#21 channels[10].rValue <= #20
#22 MOVE(oil_temp_05)
#23 channels[11].rValue <= #22
#24 MOVE(oil_temp_06)
#25 channels[12].rValue <= #24
#26 MOVE(oil_temp_07)
#27 channels[13].rValue <= #26
#28 MOVE(oil_temp_08)
#29 channels[14].rValue <= #28
#30 MOVE(oil_temp_09)
#31 channels[15].rValue <= #30
#32 MOVE(oil_temp_10)
#33 channels[16].rValue <= #32
#34 MOVE(oil_pump_01_set)
#35 channels[18].rValue <= #34
#36 MOVE(oil_pump_01_value)
#37 channels[19].rValue <= #36
#38 MOVE(oil_flow_01_value)
#39 channels[20].rValue <= #38
#40 MOVE(oil_flow_02_value)
#41 channels[21].rValue <= #40
#42 MOVE(water_temp_01)
#43 channels[22].rValue <= #42
#44 MOVE(water_temp_02)
#45 channels[23].rValue <= #44
#46 MOVE(water_temp_03)
#47 channels[24].rValue <= #46
#48 MOVE(water_temp_04)
#49 channels[25].rValue <= #48
#50 MOVE(water_temp_05)
#51 channels[26].rValue <= #50
#52 MOVE(water_temp_06)
#53 channels[27].rValue <= #52
#54 MOVE(water_temp_07)
#55 channels[28].rValue <= #54
#56 MOVE(water_temp_08)
#57 channels[29].rValue <= #56
#58 MOVE(water_temp_09)
#59 channels[30].rValue <= #58
#60 MOVE(water_temp_10)
#61 channels[31].rValue <= #60
#62 MOVE(water_pump_01_set)
#63 channels[32].rValue <= #62
#64 MOVE(water_pump_02_set)
#65 channels[33].rValue <= #64
#66 MOVE(water_flow_01_value)
#67 channels[34].rValue <= #66
#68 MOVE(air_fan_01_set)
#69 channels[35].rValue <= #68
#70 MOVE(air_fan_01_value)
#71 channels[36].rValue <= #70
#72 MOVE(air_fan_02_set)
#73 channels[37].rValue <= #72
#74 MOVE(air_fan_02_value)
#75 channels[38].rValue <= #74
#76 MOVE(water_temp_11)
#77 channels[39].rValue <= #76
_END_CFC_
(* the same logic as Structured Text *)
init();
Datalogger_01(xStart, bDtype, xTrigger, settings, channels);
channels[1].rValue := flue_gas_temp_01;
channels[2].rValue := flue_gas_temp_02;
channels[3].rValue := flue_gas_temp_03;
channels[4].rValue := flue_gas_temp_04;
channels[5].rValue := flue_gas_temp_05;
channels[6].rValue := flue_gas_temp_06;
channels[7].rValue := oil_temp_01;
channels[8].rValue := oil_temp_02;
channels[9].rValue := oil_temp_03;
channels[10].rValue := oil_temp_04;
channels[11].rValue := oil_temp_05;
channels[12].rValue := oil_temp_06;
channels[13].rValue := oil_temp_07;
channels[14].rValue := oil_temp_08;
channels[15].rValue := oil_temp_09;
channels[16].rValue := oil_temp_10;
channels[18].rValue := oil_pump_01_set;
channels[19].rValue := oil_pump_01_value;
channels[20].rValue := oil_flow_01_value;
channels[21].rValue := oil_flow_02_value;
channels[22].rValue := water_temp_01;
channels[23].rValue := water_temp_02;
channels[24].rValue := water_temp_03;
channels[25].rValue := water_temp_04;
channels[26].rValue := water_temp_05;
channels[27].rValue := water_temp_06;
channels[28].rValue := water_temp_07;
channels[29].rValue := water_temp_08;
channels[30].rValue := water_temp_09;
channels[31].rValue := water_temp_10;
channels[32].rValue := water_pump_01_set;
channels[33].rValue := water_pump_02_set;
channels[34].rValue := water_flow_01_value;
channels[35].rValue := air_fan_01_set;
channels[36].rValue := air_fan_01_value;
channels[37].rValue := air_fan_02_set;
channels[38].rValue := air_fan_02_value;
channels[39].rValue := water_temp_11;
END_PROGRAM
ACTION init:
IF xFirstCycle THEN

	settings.bInterval					:= 3;
	settings.iIntervalFactor			:= 1;
	settings.sFilename				:= 'Logfile.csv';
	settings.sPath						:= '/home/codesys_root/';
	settings.xAppendDate			:= FALSE;
	settings.xCyclicLogging			:= FALSE;
	settings.sDecimalSeparator		:=',';
	settings.sColumnSeparator		:=';';

(* Will be executed only once after start of program to enable editable channel variables *)
	(*Set all Channels to false*)
	FOR i:=1 TO 80 DO
		Channels[i].xChannelExists	:= FALSE;
	END_FOR

	Channels[1].xChannelExists		:= TRUE;
	Channels[1].sChannelName		:= 'Flue gas temperature 01';
	Channels[1].sUnit					:= '°C';
	Channels[1].rLowerLimit			:= 0;
	Channels[1].rUpperLimit			:= 400;
	Channels[1].bDecimalPlaces	:= 1;			(* number of digits afer decimal-point. IF not specified: Default-Value = 2 *)
	Channels[1].xLogAlarm			:= FALSE;		(* Shows alarm column of sine-function in file (for Standard-Datalogger) *)

	Channels[2].xChannelExists		:= TRUE;
	Channels[2].sChannelName		:= 'Flue gas temperature 02';
	Channels[2].sUnit					:= '°C';
	Channels[2].rLowerLimit			:= 0;
	Channels[2].rUpperLimit			:= 1200;
	Channels[2].bDecimalPlaces	:= 1;			(* number of digits afer decimal-point. IF not specified: Default-Value = 2 *)
	Channels[2].xLogAlarm			:= FALSE;		(* Shows alarm column of sine-function in file (for Standard-Datalogger) *)

	Channels[3].xChannelExists		:= TRUE;
	Channels[3].sChannelName		:= 'Flue gas temperature 03';
	Channels[3].sUnit					:= '°C';
	Channels[3].rLowerLimit			:= 0;
	Channels[3].rUpperLimit			:= 1200;
	Channels[3].bDecimalPlaces	:= 1;			(* number of digits afer decimal-point. IF not specified: Default-Value = 2 *)
	Channels[3].xLogAlarm			:= FALSE;		(* Shows alarm column of sine-function in file (for Standard-Datalogger) *)

	Channels[4].xChannelExists		:= TRUE;
	Channels[4].sChannelName		:= 'Flue gas temperature 04';
	Channels[4].sUnit					:= '°C';
	Channels[4].rLowerLimit			:= 0;
	Channels[4].rUpperLimit			:= 1200;
	Channels[4].bDecimalPlaces	:= 1;			(* number of digits afer decimal-point. IF not specified: Default-Value = 2 *)
	Channels[4].xLogAlarm			:= FALSE;		(* Shows alarm column of sine-function in file (for Standard-Datalogger) *)

	Channels[5].xChannelExists		:= TRUE;
	Channels[5].sChannelName		:= 'Flue gas temperature 05';
	Channels[5].sUnit					:= '°C';
	Channels[5].rLowerLimit			:= 0;
	Channels[5].rUpperLimit			:= 1200;
	Channels[5].bDecimalPlaces	:= 1;			(* number of digits afer decimal-point. IF not specified: Default-Value = 2 *)
	Channels[5].xLogAlarm			:= FALSE;		(* Shows alarm column of sine-function in file (for Standard-Datalogger) *)


	Channels[6].xChannelExists		:= TRUE;
	Channels[6].sChannelName		:= 'Flue gas temperature 06';
	Channels[6].sUnit					:= '°C';
	Channels[6].rLowerLimit			:= 0;
	Channels[6].rUpperLimit			:= 1200;
	Channels[6].bDecimalPlaces	:= 1;			(* number of digits afer decimal-point. IF not specified: Default-Value = 2 *)
	Channels[6].xLogAlarm			:= FALSE;		(* Shows alarm column of sine-function in file (for Standard-Datalogger) *)

	Channels[7].xChannelExists		:= TRUE;
	Channels[7].sChannelName		:= 'Oil temperature 01';
	Channels[7].sUnit					:= '°C';
	Channels[7].rLowerLimit			:= 0;
	Channels[7].rUpperLimit			:= 300;
	Channels[7].bDecimalPlaces	:= 1;			(* number of digits afer decimal-point. IF not specified: Default-Value = 2 *)
	Channels[7].xLogAlarm			:= FALSE;		(* Shows alarm column of sine-function in file (for Standard-Datalogger) *)

	Channels[8].xChannelExists		:= TRUE;
	Channels[8].sChannelName		:= 'Oil temperature 02';
	Channels[8].sUnit					:= '°C';
	Channels[8].rLowerLimit			:= 0;
	Channels[8].rUpperLimit			:= 300;
	Channels[8].bDecimalPlaces	:= 1;			(* number of digits afer decimal-point. IF not specified: Default-Value = 2 *)
	Channels[8].xLogAlarm			:= FALSE;		(* Shows alarm column of sine-function in file (for Standard-Datalogger) *)

	Channels[9].xChannelExists		:= TRUE;
	Channels[9].sChannelName		:= 'Oil temperature 03';
	Channels[9].sUnit					:= '°C';
	Channels[9].rLowerLimit			:= 0;
	Channels[9].rUpperLimit			:= 300;
	Channels[9].bDecimalPlaces	:= 1;			(* number of digits afer decimal-point. IF not specified: Default-Value = 2 *)
	Channels[9].xLogAlarm			:= FALSE;		(* Shows alarm column of sine-function in file (for Standard-Datalogger) *)

	Channels[10].xChannelExists		:= TRUE;
	Channels[10].sChannelName		:= 'Oil temperature 04';
	Channels[10].sUnit					:= '°C';
	Channels[10].rLowerLimit			:= 0;
	Channels[10].rUpperLimit			:= 300;
	Channels[10].bDecimalPlaces		:= 1;			(* number of digits afer decimal-point. IF not specified: Default-Value = 2 *)
	Channels[10].xLogAlarm				:= FALSE;		(* Shows alarm column of sine-function in file (for Standard-Datalogger) *)

	Channels[11].xChannelExists		:= TRUE;
	Channels[11].sChannelName		:= 'Oil temperature 05';
	Channels[11].sUnit					:= '°C';
	Channels[11].rLowerLimit			:= 0;
	Channels[11].rUpperLimit			:= 300;
	Channels[11].bDecimalPlaces		:= 1;			(* number of digits afer decimal-point. IF not specified: Default-Value = 2 *)
	Channels[11].xLogAlarm				:= FALSE;		(* Shows alarm column of sine-function in file (for Standard-Datalogger) *)

	Channels[12].xChannelExists		:= TRUE;
	Channels[12].sChannelName		:= 'Oil temperature 06';
	Channels[12].sUnit					:= '°C';
	Channels[12].rLowerLimit			:= 0;
	Channels[12].rUpperLimit			:= 300;
	Channels[12].bDecimalPlaces		:= 1;			(* number of digits afer decimal-point. IF not specified: Default-Value = 2 *)
		Channels[12].xLogAlarm			:= FALSE;		(* Shows alarm column of sine-function in file (for Standard-Datalogger) *)

	Channels[13].xChannelExists		:= TRUE;
	Channels[13].sChannelName		:= 'Oil temperature 07';
	Channels[13].sUnit					:= '°C';
	Channels[13].rLowerLimit			:= 0;
	Channels[13].rUpperLimit			:= 300;
	Channels[13].bDecimalPlaces		:= 1;			(* number of digits afer decimal-point. IF not specified: Default-Value = 2 *)
	Channels[13].xLogAlarm				:= FALSE;		(* Shows alarm column of sine-function in file (for Standard-Datalogger) *)

	Channels[14].xChannelExists		:= TRUE;
	Channels[14].sChannelName		:= 'Oil temperature 08';
	Channels[14].sUnit					:= '°C';
	Channels[14].rLowerLimit			:= 0;
	Channels[14].rUpperLimit			:= 300;
	Channels[14].bDecimalPlaces		:= 1;			(* number of digits afer decimal-point. IF not specified: Default-Value = 2 *)
	Channels[14].xLogAlarm				:= FALSE;		(* Shows alarm column of sine-function in file (for Standard-Datalogger) *)

	Channels[15].xChannelExists		:= TRUE;
	Channels[15].sChannelName		:= 'Oil temperature 09';
	Channels[15].sUnit					:= '°C';
	Channels[15].rLowerLimit			:= 0;
	Channels[15].rUpperLimit			:= 300;
	Channels[15].bDecimalPlaces		:= 1;			(* number of digits afer decimal-point. IF not specified: Default-Value = 2 *)
		Channels[15].xLogAlarm			:= FALSE;		(* Shows alarm column of sine-function in file (for Standard-Datalogger) *)

	Channels[16].xChannelExists		:= TRUE;
	Channels[16].sChannelName		:= 'Oil temperature 10';
	Channels[16].sUnit					:= '°C';
	Channels[16].rLowerLimit			:= 0;
	Channels[16].rUpperLimit			:= 300;
	Channels[16].bDecimalPlaces		:= 1;			(* number of digits afer decimal-point. IF not specified: Default-Value = 2 *)
	Channels[16].xLogAlarm				:= FALSE;		(* Shows alarm column of sine-function in file (for Standard-Datalogger) *)

	Channels[17].xChannelExists		:= TRUE;
	Channels[17].sChannelName		:= 'Oil temperature 11';
	Channels[17].sUnit					:= '°C';
	Channels[17].rLowerLimit			:= 0;
	Channels[17].rUpperLimit			:= 300;
	Channels[17].bDecimalPlaces		:= 1;			(* number of digits afer decimal-point. IF not specified: Default-Value = 2 *)
	Channels[17].xLogAlarm				:= FALSE;		(* Shows alarm column of sine-function in file (for Standard-Datalogger) *)

	Channels[18].xChannelExists		:= TRUE;
	Channels[18].sChannelName		:= 'Oil pump set';
	Channels[18].sUnit					:= '%';
	Channels[18].rLowerLimit			:= 0;
	Channels[18].rUpperLimit			:= 100;
	Channels[18].bDecimalPlaces		:= 1;			(* number of digits afer decimal-point. IF not specified: Default-Value = 2 *)
	Channels[18].xLogAlarm				:= FALSE;		(* Shows alarm column of sine-function in file (for Standard-Datalogger) *)

	Channels[19].xChannelExists		:= TRUE;
	Channels[19].sChannelName		:= 'Oil pump speed';
	Channels[19].sUnit					:= '%';
	Channels[19].rLowerLimit			:= 0;
	Channels[19].rUpperLimit			:= 100;
	Channels[19].bDecimalPlaces		:= 1;			(* number of digits afer decimal-point. IF not specified: Default-Value = 2 *)
	Channels[19].xLogAlarm				:= FALSE;		(* Shows alarm column of sine-function in file (for Standard-Datalogger) *)

	Channels[20].xChannelExists		:= TRUE;
	Channels[20].sChannelName		:= 'Oil flow 01';
	Channels[20].sUnit					:= 'dm3/min';
	Channels[20].rLowerLimit			:= 0;
	Channels[20].rUpperLimit			:= 100;
	Channels[20].bDecimalPlaces		:= 1;			(* number of digits afer decimal-point. IF not specified: Default-Value = 2 *)
	Channels[20].xLogAlarm				:= FALSE;		(* Shows alarm column of sine-function in file (for Standard-Datalogger) *)

	Channels[21].xChannelExists		:= TRUE;
	Channels[21].sChannelName		:= 'Oil flow 02';
	Channels[21].sUnit					:= 'dm3/min';
	Channels[21].rLowerLimit			:= 0;
	Channels[21].rUpperLimit			:= 100;
	Channels[21].bDecimalPlaces		:= 1;			(* number of digits afer decimal-point. IF not specified: Default-Value = 2 *)
	Channels[21].xLogAlarm				:= FALSE;		(* Shows alarm column of sine-function in file (for Standard-Datalogger) *)

	Channels[22].xChannelExists		:= TRUE;
	Channels[22].sChannelName		:= 'Water temperature 01';
	Channels[22].sUnit					:= '°C';
	Channels[22].rLowerLimit			:= 0;
	Channels[22].rUpperLimit			:= 100;
	Channels[22].bDecimalPlaces		:= 1;			(* number of digits afer decimal-point. IF not specified: Default-Value = 2 *)
	Channels[22].xLogAlarm				:= FALSE;		(* Shows alarm column of sine-function in file (for Standard-Datalogger) *)

	Channels[23].xChannelExists		:= TRUE;
	Channels[23].sChannelName		:= 'Water temperature 02';
	Channels[23].sUnit					:= '°C';
	Channels[23].rLowerLimit			:= 0;
	Channels[23].rUpperLimit			:= 100;
	Channels[23].bDecimalPlaces		:= 1;			(* number of digits afer decimal-point. IF not specified: Default-Value = 2 *)
	Channels[23].xLogAlarm				:= FALSE;		(* Shows alarm column of sine-function in file (for Standard-Datalogger) *)

	Channels[24].xChannelExists		:= TRUE;
	Channels[24].sChannelName		:= 'Water temperature 03';
	Channels[24].sUnit					:= '°C';
	Channels[24].rLowerLimit			:= 0;
	Channels[24].rUpperLimit			:= 100;
	Channels[24].bDecimalPlaces		:= 1;			(* number of digits afer decimal-point. IF not specified: Default-Value = 2 *)
	Channels[24].xLogAlarm				:= FALSE;		(* Shows alarm column of sine-function in file (for Standard-Datalogger) *)

	Channels[25].xChannelExists		:= TRUE;
	Channels[25].sChannelName		:= 'Water temperature 04';
	Channels[25].sUnit					:= '°C';
	Channels[25].rLowerLimit			:= 0;
	Channels[25].rUpperLimit			:= 100;
	Channels[25].bDecimalPlaces		:= 1;			(* number of digits afer decimal-point. IF not specified: Default-Value = 2 *)
	Channels[25].xLogAlarm				:= FALSE;		(* Shows alarm column of sine-function in file (for Standard-Datalogger) *)

	Channels[26].xChannelExists		:= TRUE;
	Channels[26].sChannelName		:= 'Water temperature 05';
	Channels[26].sUnit					:= '°C';
	Channels[26].rLowerLimit			:= 0;
	Channels[26].rUpperLimit			:= 100;
	Channels[26].bDecimalPlaces		:= 1;			(* number of digits afer decimal-point. IF not specified: Default-Value = 2 *)
	Channels[26].xLogAlarm				:= FALSE;		(* Shows alarm column of sine-function in file (for Standard-Datalogger) *)

	Channels[27].xChannelExists		:= TRUE;
	Channels[27].sChannelName		:= 'Water temperature 06';
	Channels[27].sUnit					:= '°C';
	Channels[27].rLowerLimit			:= 0;
	Channels[27].rUpperLimit			:= 100;
	Channels[27].bDecimalPlaces		:= 1;			(* number of digits afer decimal-point. IF not specified: Default-Value = 2 *)
	Channels[27].xLogAlarm				:= FALSE;		(* Shows alarm column of sine-function in file (for Standard-Datalogger) *)

	Channels[28].xChannelExists		:= TRUE;
	Channels[28].sChannelName		:= 'Water temperature 07';
	Channels[28].sUnit					:= '°C';
	Channels[28].rLowerLimit			:= 0;
	Channels[28].rUpperLimit			:= 100;
	Channels[28].bDecimalPlaces		:= 1;			(* number of digits afer decimal-point. IF not specified: Default-Value = 2 *)
	Channels[28].xLogAlarm				:= FALSE;		(* Shows alarm column of sine-function in file (for Standard-Datalogger) *)

	Channels[29].xChannelExists		:= TRUE;
	Channels[29].sChannelName		:= 'Water temperature 08';
	Channels[29].sUnit					:= '°C';
	Channels[29].rLowerLimit			:= 0;
	Channels[29].rUpperLimit			:= 100;
	Channels[29].bDecimalPlaces		:= 1;			(* number of digits afer decimal-point. IF not specified: Default-Value = 2 *)
	Channels[29].xLogAlarm				:= FALSE;		(* Shows alarm column of sine-function in file (for Standard-Datalogger) *)

	Channels[30].xChannelExists		:= TRUE;
	Channels[30].sChannelName		:= 'Water temperature 09';
	Channels[30].sUnit					:= '°C';
	Channels[30].rLowerLimit			:= 0;
	Channels[30].rUpperLimit			:= 100;
	Channels[30].bDecimalPlaces		:= 1;			(* number of digits afer decimal-point. IF not specified: Default-Value = 2 *)
	Channels[30].xLogAlarm				:= FALSE;		(* Shows alarm column of sine-function in file (for Standard-Datalogger) *)

	Channels[31].xChannelExists		:= TRUE;
	Channels[31].sChannelName		:= 'Water temperature 10';
	Channels[31].sUnit					:= '°C';
	Channels[31].rLowerLimit			:= 0;
	Channels[31].rUpperLimit			:= 100;
	Channels[31].bDecimalPlaces		:= 1;			(* number of digits afer decimal-point. IF not specified: Default-Value = 2 *)
	Channels[31].xLogAlarm				:= FALSE;		(* Shows alarm column of sine-function in file (for Standard-Datalogger) *)

	Channels[32].xChannelExists		:= TRUE;
	Channels[32].sChannelName		:= 'Water pump 01 set';
	Channels[32].sUnit					:= '%';
	Channels[32].rLowerLimit			:= 0;
	Channels[32].rUpperLimit			:= 100;
	Channels[32].bDecimalPlaces		:= 1;			(* number of digits afer decimal-point. IF not specified: Default-Value = 2 *)
	Channels[32].xLogAlarm				:= FALSE;		(* Shows alarm column of sine-function in file (for Standard-Datalogger) *)

	Channels[33].xChannelExists		:= TRUE;
	Channels[33].sChannelName		:= 'Water pump 02 set';
	Channels[33].sUnit					:= '%';
	Channels[33].rLowerLimit			:= 0;
	Channels[33].rUpperLimit			:= 100;
	Channels[33].bDecimalPlaces		:= 1;			(* number of digits afer decimal-point. IF not specified: Default-Value = 2 *)
	Channels[33].xLogAlarm				:= FALSE;		(* Shows alarm column of sine-function in file (for Standard-Datalogger) *)

	Channels[34].xChannelExists		:= TRUE;
	Channels[34].sChannelName		:= 'Water flow';
	Channels[34].sUnit					:= 'm3/h';
	Channels[34].rLowerLimit			:= 0;
	Channels[34].rUpperLimit			:= 100;
	Channels[34].bDecimalPlaces		:= 1;			(* number of digits afer decimal-point. IF not specified: Default-Value = 2 *)
	Channels[34].xLogAlarm				:= FALSE;		(* Shows alarm column of sine-function in file (for Standard-Datalogger) *)

	Channels[35].xChannelExists		:= TRUE;
	Channels[35].sChannelName		:= 'Inlet air fan set';
	Channels[35].sUnit					:= '%';
	Channels[35].rLowerLimit			:= 0;
	Channels[35].rUpperLimit			:= 100;
	Channels[35].bDecimalPlaces		:= 1;			(* number of digits afer decimal-point. IF not specified: Default-Value = 2 *)
	Channels[35].xLogAlarm				:= FALSE;		(* Shows alarm column of sine-function in file (for Standard-Datalogger) *)

	Channels[36].xChannelExists		:= TRUE;
	Channels[36].sChannelName		:= 'Inlet air fan speed';
	Channels[36].sUnit					:= '%';
	Channels[36].rLowerLimit			:= 0;
	Channels[36].rUpperLimit			:= 100;
	Channels[36].bDecimalPlaces		:= 1;			(* number of digits afer decimal-point. IF not specified: Default-Value = 2 *)
	Channels[36].xLogAlarm				:= FALSE;		(* Shows alarm column of sine-function in file (for Standard-Datalogger) *)

	Channels[37].xChannelExists		:= TRUE;
	Channels[37].sChannelName		:= 'Outlet air fan set';
	Channels[37].sUnit					:= '%';
	Channels[37].rLowerLimit			:= 0;
	Channels[37].rUpperLimit			:= 100;
	Channels[37].bDecimalPlaces		:= 1;			(* number of digits afer decimal-point. IF not specified: Default-Value = 2 *)
	Channels[37].xLogAlarm				:= FALSE;		(* Shows alarm column of sine-function in file (for Standard-Datalogger) *)

	Channels[38].xChannelExists		:= TRUE;
	Channels[38].sChannelName		:= 'Outlet air fan speed';
	Channels[38].sUnit					:= '%';
	Channels[38].rLowerLimit			:= 0;
	Channels[38].rUpperLimit			:= 100;
	Channels[38].bDecimalPlaces		:= 1;			(* number of digits afer decimal-point. IF not specified: Default-Value = 2 *)
	Channels[38].xLogAlarm				:= FALSE;		(* Shows alarm column of sine-function in file (for Standard-Datalogger) *)

	Channels[39].xChannelExists		:= TRUE;
	Channels[39].sChannelName		:= 'Water temperature 10';
	Channels[39].sUnit					:= '°C';
	Channels[39].rLowerLimit			:= 0;
	Channels[39].rUpperLimit			:= 100;
	Channels[39].bDecimalPlaces		:= 1;			(* number of digits afer decimal-point. IF not specified: Default-Value = 2 *)
	Channels[39].xLogAlarm				:= FALSE;		(* Shows alarm column of sine-function in file (for Standard-Datalogger) *)

	xFirstCycle						:= FALSE;		(* Prevents another call of initialization *)

END_IF


(* Entries outside of IF-THEN construct will be executed in each cycle of the PLC *)
END_ACTION

(* POU timer, LD *)
FUNCTION_BLOCK timer
VAR_INPUT
	interval: TIME;
	start_timer: BOOL;
END_VAR
VAR_OUTPUT
END_VAR
VAR
	ton_01: TON;
	ton_02: TON;
END_VAR
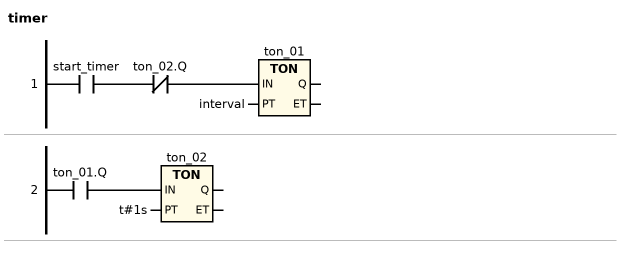
_LD_ (* Ladder Diagram *)
NETWORK 1
	[start_timer] - [/ton_02.Q] - ton_01:TON(IN: *, PT: interval)
NETWORK 2
	[ton_01.Q] - ton_02:TON(IN: *, PT: t#1s)
_END_LD_
(* the same logic as Structured Text *)
(* Network 1 *)
ton_01(IN := start_timer AND NOT ton_02.Q, PT := interval);
(* Network 2 *)
ton_02(IN := ton_01.Q, PT := t#1s);
END_FUNCTION_BLOCK

(* Visualisation Channel_VISU
embedded screen at (10,0)-(801,551): Channel_VISU_Basic
*)

(* Visualisation Logger_VISU
embedded screen at (10,10)-(821,571): Logger_VISU_Basic
*)

(* Visualisation PLC_VISU
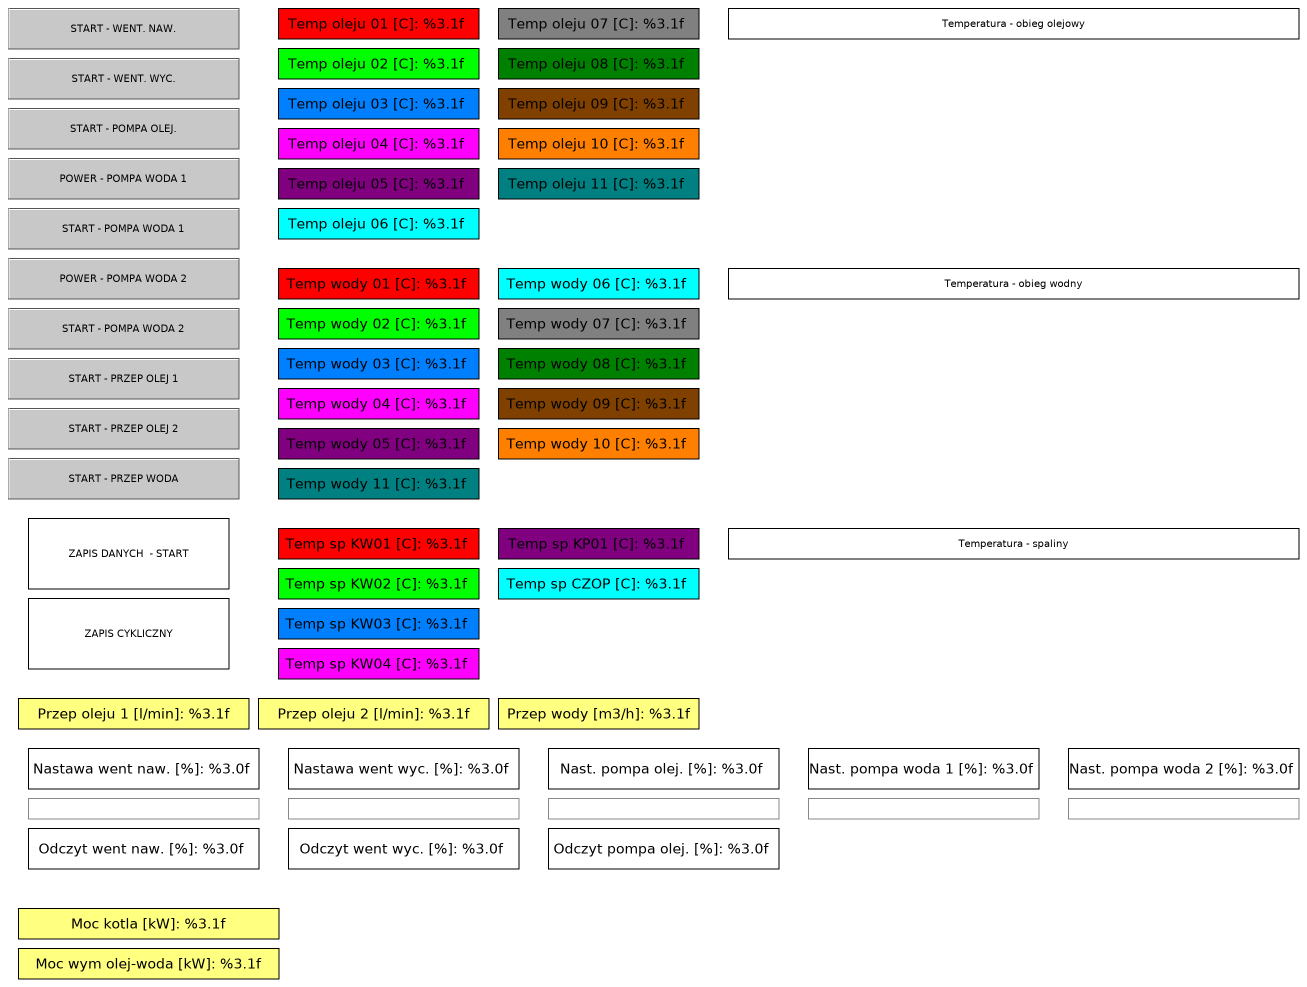
rectangle at (30,520)-(231,591): text "ZAPIS DANYCH  - START"; toggles SAVE_DATA.xStart
button at (10,10)-(241,51): text "START - WENT. NAW."; toggles .air_fan_01_start
button at (10,60)-(241,101): text "START - WENT. WYC."; toggles .air_fan_02_start
button at (10,110)-(241,151): text "START - POMPA OLEJ."; toggles .oil_pump_01_start
button at (10,210)-(241,251): text "START - POMPA WODA 1"; toggles .water_pump_01_start
button at (10,310)-(241,351): text "START - POMPA WODA 2"; toggles .water_pump_02_start
button at (10,160)-(241,201): text "POWER - POMPA WODA 1"; toggles .water_pump_01_power
button at (10,260)-(241,301): text "POWER - POMPA WODA 2"; toggles .water_pump_02_power
button at (10,360)-(241,401): text "START - PRZEP OLEJ 1"; toggles .oil_flow_01_start
button at (10,410)-(241,451): text "START - PRZEP OLEJ 2"; toggles .oil_flow_02_start
button at (10,460)-(241,501): text "START - PRZEP WODA"; toggles .water_flow_01_start
rectangle at (280,10)-(481,41): text "Temp oleju 01 [C]: %3.1f"; shows .oil_temp_01
rectangle at (280,50)-(481,81): text "Temp oleju 02 [C]: %3.1f"; shows .oil_temp_02
rectangle at (280,90)-(481,121): text "Temp oleju 03 [C]: %3.1f"; shows .oil_temp_03
rectangle at (280,130)-(481,161): text "Temp oleju 04 [C]: %3.1f"; shows .oil_temp_04
rectangle at (280,170)-(481,201): text "Temp oleju 05 [C]: %3.1f"; shows .oil_temp_05
rectangle at (280,210)-(481,241): text "Temp oleju 06 [C]: %3.1f"; shows .oil_temp_06
rectangle at (500,10)-(701,41): text "Temp oleju 07 [C]: %3.1f"; shows .oil_temp_07
rectangle at (500,50)-(701,81): text "Temp oleju 08 [C]: %3.1f"; shows .oil_temp_08
rectangle at (500,90)-(701,121): text "Temp oleju 09 [C]: %3.1f"; shows .oil_temp_09
rectangle at (500,130)-(701,161): text "Temp oleju 10 [C]: %3.1f"; shows .oil_temp_10
rectangle at (500,170)-(701,201): text "Temp oleju 11 [C]: %3.1f"; shows .oil_temp_11
rectangle at (280,270)-(481,301): text "Temp wody 01 [C]: %3.1f"; shows .water_temp_01
rectangle at (280,310)-(481,341): text "Temp wody 02 [C]: %3.1f"; shows .water_temp_02
rectangle at (280,350)-(481,381): text "Temp wody 03 [C]: %3.1f"; shows .water_temp_03
rectangle at (280,390)-(481,421): text "Temp wody 04 [C]: %3.1f"; shows .water_temp_04
rectangle at (280,430)-(481,461): text "Temp wody 05 [C]: %3.1f"; shows .water_temp_05
rectangle at (500,270)-(701,301): text "Temp wody 06 [C]: %3.1f"; shows .water_temp_06
rectangle at (500,310)-(701,341): text "Temp wody 07 [C]: %3.1f"; shows .water_temp_07
rectangle at (500,350)-(701,381): text "Temp wody 08 [C]: %3.1f"; shows .water_temp_08
rectangle at (500,390)-(701,421): text "Temp wody 09 [C]: %3.1f"; shows .water_temp_09
rectangle at (500,430)-(701,461): text "Temp wody 10 [C]: %3.1f"; shows .water_temp_10
rectangle at (30,750)-(261,791): text "Nastawa went naw. [%]: %3.0f"; shows .air_fan_01_set; editable 0..100
rectangle at (30,830)-(261,871): text "Odczyt went naw. [%]: %3.0f"; shows .air_fan_01_value
rectangle at (290,750)-(521,791): text "Nastawa went wyc. [%]: %3.0f"; shows .air_fan_02_set; editable 0..100
rectangle at (290,830)-(521,871): text "Odczyt went wyc. [%]: %3.0f"; shows .air_fan_02_value
rectangle at (550,750)-(781,791): text "Nast. pompa olej. [%]: %3.0f"; shows .oil_pump_01_set; editable 0..100
rectangle at (550,830)-(781,871): text "Odczyt pompa olej. [%]: %3.0f"; shows .oil_pump_01_value
rectangle at (810,750)-(1041,791): text "Nast. pompa woda 1 [%]: %3.0f"; shows .water_pump_01_set; editable 0..100
rectangle at (1070,750)-(1301,791): text "Nast. pompa woda 2 [%]: %3.0f"; shows .water_pump_02_set; editable 0..100
rectangle at (730,10)-(1301,41): text "Temperatura - obieg olejowy"
rectangle at (730,270)-(1301,301): text "Temperatura - obieg wodny"
rectangle at (730,530)-(1301,561): text "Temperatura - spaliny"
rectangle at (280,530)-(481,561): text "Temp sp KW01 [C]: %3.1f"; shows .flue_gas_temp_02
rectangle at (280,570)-(481,601): text "Temp sp KW02 [C]: %3.1f"; shows .flue_gas_temp_03
rectangle at (280,610)-(481,641): text "Temp sp KW03 [C]: %3.1f"; shows .flue_gas_temp_04
rectangle at (280,650)-(481,681): text "Temp sp KW04 [C]: %3.1f"; shows .flue_gas_temp_05
rectangle at (500,530)-(701,561): text "Temp sp KP01 [C]: %3.1f"; shows .flue_gas_temp_06
rectangle at (500,570)-(701,601): text "Temp sp CZOP [C]: %3.1f"; shows .flue_gas_temp_01
rectangle at (280,470)-(481,501): text "Temp wody 11 [C]: %3.1f"; shows .water_temp_11
rectangle at (20,700)-(251,731): text "Przep oleju 1 [l/min]: %3.1f"; shows .oil_flow_01_value
rectangle at (260,700)-(491,731): text "Przep oleju 2 [l/min]: %3.1f"; shows .oil_flow_02_value
rectangle at (500,700)-(701,731): text "Przep wody [m3/h]: %3.1f"; shows .water_flow_01_value
rectangle at (30,600)-(231,671): text "ZAPIS CYKLICZNY"; toggles SAVE_DATA.settings.xCyclicLogging
rectangle at (20,910)-(281,941): text "Moc kotla [kW]: %3.1f"; shows PLC_PRG.Boiler_Power.OIL_POWER
rectangle at (20,950)-(281,981): text "Moc wym olej-woda [kW]: %3.1f"; shows PLC_PRG.Oil_Water_Heat_Exchanger_Power.OIL_POWER
5 more shapes without text or variables
4 elements of other kinds (tables, trends, ...) not read
*)

(* Visualisation PLC_VISU_OIL
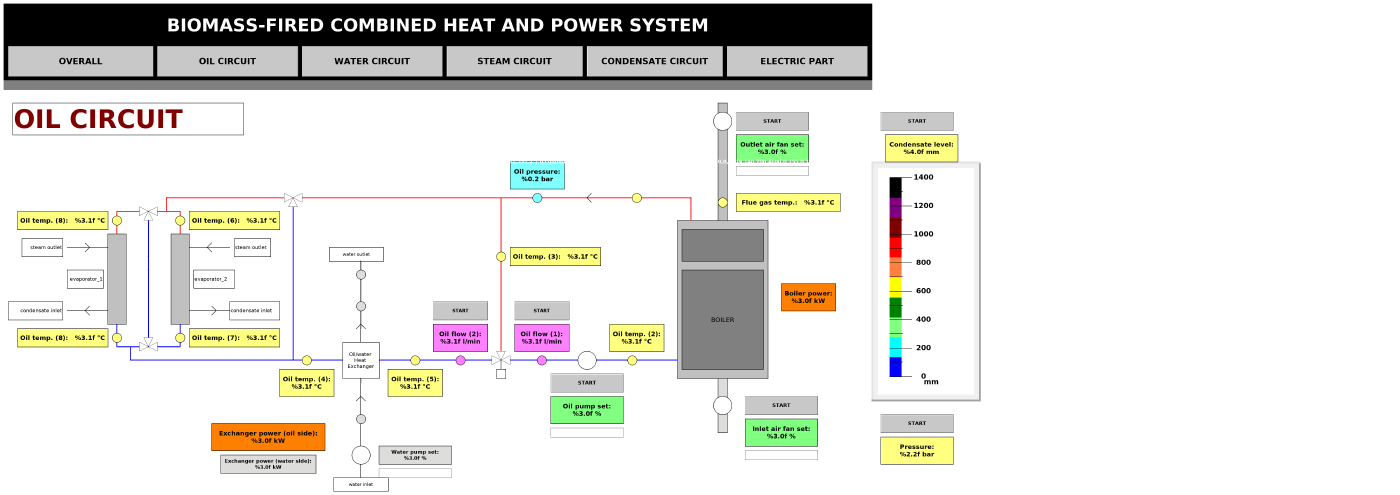
rectangle at (1500,590)-(1681,811): text "BOILER"
rectangle at (750,750)-(831,831): text "Oil/water / Heat / Exchanger"
rectangle at (30,460)-(231,501): text "Oil temp. (8):   %3.1f °C"; shows .oil_temp_08
rectangle at (1210,870)-(1371,931): text "Oil pump set: / %3.0f %"; shows .oil_pump_01_set; editable 20..100
rectangle at (950,710)-(1071,771): text "Oil flow (2): / %3.1f l/min"; shows .oil_flow_02_value
rectangle at (20,220)-(531,291): text "OIL CIRCUIT"
rectangle at (730,1050)-(851,1081): text "water inlet"
rectangle at (720,540)-(841,571): text "water outlet"
rectangle at (1120,350)-(1241,411): text "Oil pressure: / %0.2 bar"
rectangle at (140,590)-(221,631): text "evaporator_1"
rectangle at (40,520)-(131,561): text "steam outlet"
rectangle at (10,660)-(131,701): text "condensate inlet"
rectangle at (420,590)-(511,631): text "evaporator_2"
rectangle at (510,520)-(591,561): text "steam outlet"
rectangle at (500,660)-(611,701): text "condensate inlet"
rectangle at (30,720)-(231,761): text "Oil temp. (8):   %3.1f °C"; shows .oil_temp_09
rectangle at (410,460)-(611,501): text "Oil temp. (6):   %3.1f °C"; shows .oil_temp_06
rectangle at (410,720)-(611,761): text "Oil temp. (7):   %3.1f °C"; shows .oil_temp_07
rectangle at (610,810)-(731,871): text "Oil temp. (4): / %3.1f °C"; shows .oil_temp_04
rectangle at (1130,710)-(1251,771): text "Oil flow (1): / %3.1f l/min"; shows .oil_flow_01_value
rectangle at (850,810)-(971,871): text "Oil temp. (5): / %3.1f °C"; shows .oil_temp_05
rectangle at (1340,710)-(1461,771): text "Oil temp. (2): / %3.1f °C"; shows .oil_temp_02
button at (1210,820)-(1371,861): text "START"; toggles .oil_pump_01_start
button at (1130,660)-(1251,701): text "START"; toggles .oil_flow_01_start
button at (950,660)-(1071,701): text "START"; toggles .oil_flow_02_start
rectangle at (1120,540)-(1321,581): text "Oil temp. (3):   %3.1f °C"; shows .oil_temp_03
button at (1620,240)-(1781,281): text "START"; toggles .air_fan_02_start
rectangle at (1620,290)-(1781,351): text "Outlet air fan set: / %3.0f %"; shows .air_fan_02_set; editable 20..100
button at (1640,870)-(1801,911): text "START"; toggles .air_fan_01_start
rectangle at (1640,920)-(1801,981): text "Inlet air fan set: / %3.0f %"; shows .air_fan_01_set; editable 30..100
rectangle at (1620,420)-(1851,461): text "Flue gas temp.:   %3.1f °C"; shows .flue_gas_temp_01
embedded screen at (0,0)-(1921,171): VISU_MENU
rectangle at (1720,620)-(1841,681): text "Boiler power: / %3.0f kW"; shows PLC_PRG.Boiler_Power.OIL_POWER
rectangle at (460,930)-(711,991): text "Exchanger power (oil side): / %3.0f kW"; shows PLC_PRG.Oil_Water_Heat_Exchanger_Oil_Side_Power.OIL_POWER
rectangle at (830,980)-(991,1021): text "Water pump set: / %3.0f %"; shows .water_pump_01_set; editable 0..100
rectangle at (480,1000)-(691,1041): text "Exchanger power (water side): / %3.0f kW"; shows PLC_PRG.Oil_Water_Heat_Exchanger_Water_Side_Power.WATER_POWER
group at (1920,350)-(2161,881)
  rectangle at (0,0)-(1,1): text "{ExtendedElement},Visu\ElementDLL.ete,1,@Bargraph,241,531,2,1,0,condensate_level_01_value,mm,%4.0f,100,200,0,1400,0,0,0,0,0,0,0,-19,140,700,Arial,0,255,0,255,0,0,0,0,0,1,10,0,140,0,0,255,140,280,0,255,255,280,420,128,255,128,420,560,0,128,0,560,700,255,255,0,700,840,255,128,64,840,980,255,0,0,980,1120,127,0,0,1120,1260,128,0,128,1260,1400,0,0,0,1,0,,0,0,0,"
  rectangle at (40,432)-(66,477): invisible if (condensate_level_01_value * 1.0) < 0; top (MIN(MAX(0, (condensate_level_01_value * 1.0)),140)  - 140)  * -0.314286
  rectangle at (40,388)-(66,433): invisible if (condensate_level_01_value * 1.0) < 140; top (MIN(MAX(140, (condensate_level_01_value * 1.0)),280)  - 280)  * -0.314286
  rectangle at (40,344)-(66,389): invisible if (condensate_level_01_value * 1.0) < 280; top (MIN(MAX(280, (condensate_level_01_value * 1.0)),420)  - 420)  * -0.314286
  rectangle at (40,300)-(66,345): invisible if (condensate_level_01_value * 1.0) < 420; top (MIN(MAX(420, (condensate_level_01_value * 1.0)),560)  - 560)  * -0.314286
  rectangle at (40,255)-(66,301): invisible if (condensate_level_01_value * 1.0) < 560; top (MIN(MAX(560, (condensate_level_01_value * 1.0)),700)  - 700)  * -0.321429
  rectangle at (40,211)-(66,256): invisible if (condensate_level_01_value * 1.0) < 700; top (MIN(MAX(700, (condensate_level_01_value * 1.0)),840)  - 840)  * -0.314286
  rectangle at (40,167)-(66,212): invisible if (condensate_level_01_value * 1.0) < 840; top (MIN(MAX(840, (condensate_level_01_value * 1.0)),980)  - 980)  * -0.314286
  rectangle at (40,123)-(66,168): invisible if (condensate_level_01_value * 1.0) < 980; top (MIN(MAX(980, (condensate_level_01_value * 1.0)),1120)  - 1120)  * -0.314286
  rectangle at (40,79)-(66,124): invisible if (condensate_level_01_value * 1.0) < 1120; top (MIN(MAX(1120, (condensate_level_01_value * 1.0)),1260)  - 1260)  * -0.314286
  rectangle at (40,35)-(66,80): invisible if (condensate_level_01_value * 1.0) < 1260; top (MIN(MAX(1260, (condensate_level_01_value * 1.0)),1400)  - 1400)  * -0.314286
  rectangle at (91,461)-(224,490): text "0"
  rectangle at (91,398)-(224,427): text "200"
  rectangle at (91,335)-(224,364): text "400"
  rectangle at (91,272)-(224,301): text "600"
  rectangle at (91,209)-(224,238): text "800"
  rectangle at (91,146)-(224,175): text "1000"
  rectangle at (91,83)-(224,112): text "1200"
  rectangle at (91,20)-(224,49): text "1400"
  rectangle at (98,477)-(166,499): text "mm"
button at (1940,240)-(2101,281): text "START"; toggles .condensate_level_01_start
rectangle at (1940,960)-(2101,1021): text "Pressure: / %2.2f bar"; shows .steam_pressure_01_value
button at (1940,910)-(2101,951): text "START"; toggles .steam_pressure_01_start
rectangle at (1950,290)-(2111,351): text "Condensate level: / %4.0f mm"; shows .condensate_level_01_value
94 more shapes without text or variables
8 elements of other kinds (tables, trends, ...) not read
*)

(* Visualisation PLC_VISU_STEAM
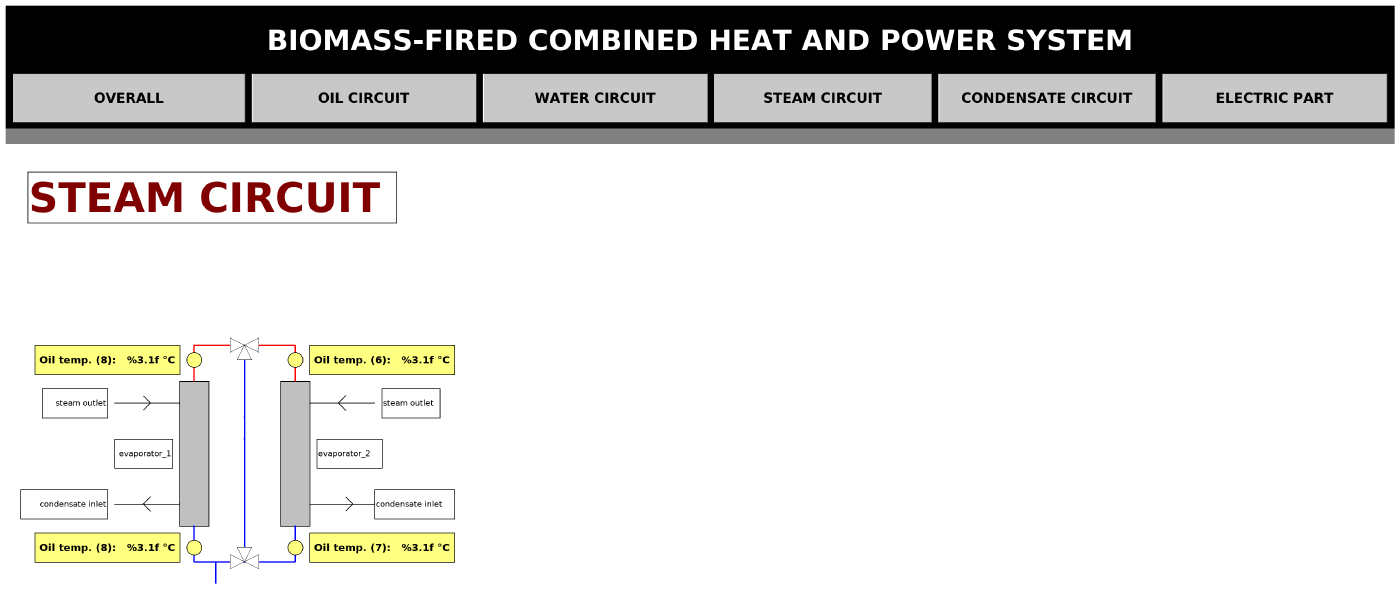
embedded screen at (0,0)-(1921,171): VISU_MENU
rectangle at (40,470)-(241,511): text "Oil temp. (8):   %3.1f °C"; shows .oil_temp_08
rectangle at (30,230)-(541,301): text "STEAM CIRCUIT"
rectangle at (150,600)-(231,641): text "evaporator_1"
rectangle at (50,530)-(141,571): text "steam outlet"
rectangle at (20,670)-(141,711): text "condensate inlet"
rectangle at (430,600)-(521,641): text "evaporator_2"
rectangle at (520,530)-(601,571): text "steam outlet"
rectangle at (510,670)-(621,711): text "condensate inlet"
rectangle at (40,730)-(241,771): text "Oil temp. (8):   %3.1f °C"; shows .oil_temp_09
rectangle at (420,470)-(621,511): text "Oil temp. (6):   %3.1f °C"; shows .oil_temp_06
rectangle at (420,730)-(621,771): text "Oil temp. (7):   %3.1f °C"; shows .oil_temp_07
29 more shapes without text or variables
*)

(* Visualisation PLC_VISU_WATER
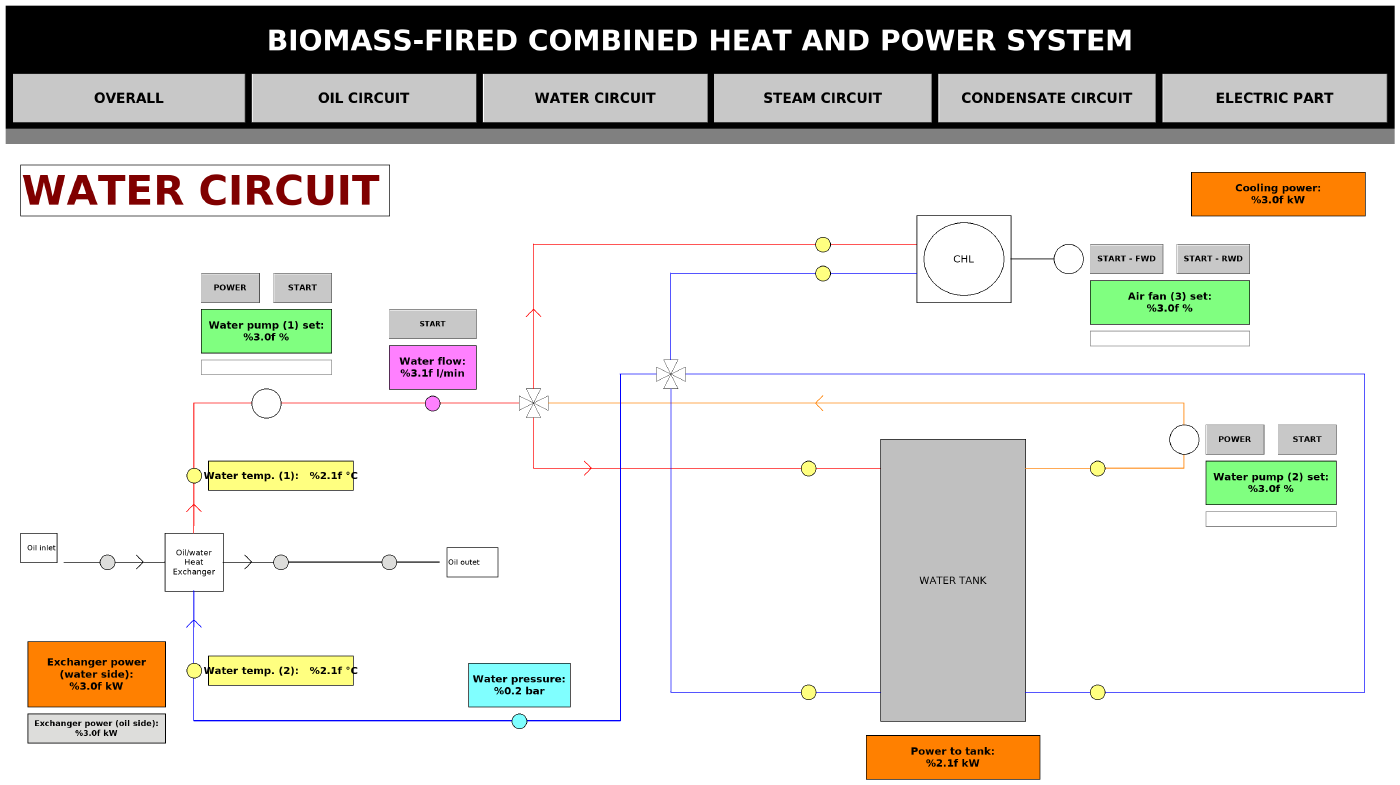
rectangle at (1210,600)-(1411,991): text "WATER TANK"
rectangle at (220,730)-(301,811): text "Oil/water / Heat / Exchanger"
rectangle at (20,730)-(71,771): text "Oil inlet"
rectangle at (610,750)-(681,791): text "Oil outet"
ellipse at (1270,300)-(1381,401): text "CHL"
embedded screen at (0,0)-(1921,171): VISU_MENU
rectangle at (20,220)-(531,291): text "WATER CIRCUIT"
button at (370,370)-(451,411): text "START"; toggles .water_pump_01_start
rectangle at (270,420)-(451,481): text "Water pump (1) set: / %3.0f %"; shows .water_pump_01_set; editable 0..100
button at (270,370)-(351,411): text "POWER"; toggles .water_pump_01_power
rectangle at (530,470)-(651,531): text "Water flow: / %3.1f l/min"; shows .water_flow_01_value
button at (530,420)-(651,461): text "START"; toggles .water_flow_01_start
rectangle at (280,630)-(481,671): text "Water temp. (1):   %2.1f °C"; shows .water_temp_01
rectangle at (280,900)-(481,941): text "Water temp. (2):   %2.1f °C"; shows .water_temp_02
rectangle at (640,910)-(781,971): text "Water pressure: / %0.2 bar"
button at (1760,580)-(1841,621): text "START"; toggles .water_pump_02_start
rectangle at (1660,630)-(1841,691): text "Water pump (2) set: / %3.0f %"; shows .water_pump_02_set; editable 0..100
button at (1660,580)-(1741,621): text "POWER"; toggles .water_pump_02_power
button at (1620,330)-(1721,371): text "START - RWD"; invisible if .air_fan_03_start_fwd; toggles .air_fan_03_start_rwd
rectangle at (1500,380)-(1721,441): text "Air fan (3) set: / %3.0f %"; shows .air_fan_03_set; editable 10..100
button at (1500,330)-(1601,371): text "START - FWD"; invisible if .air_fan_03_start_rwd; toggles .air_fan_03_start_fwd
rectangle at (30,880)-(221,971): text "Exchanger power / (water side): / %3.0f kW"; shows PLC_PRG.Oil_Water_Heat_Exchanger_Water_Side_Power.WATER_POWER
rectangle at (30,980)-(221,1021): text "Exchanger power (oil side): / %3.0f kW"; shows PLC_PRG.Oil_Water_Heat_Exchanger_Oil_Side_Power.OIL_POWER
rectangle at (1190,1010)-(1431,1071): text "Power to tank: / %2.1f kW"; shows PLC_PRG.Tank_Power.WATER_POWER
rectangle at (1640,230)-(1881,291): text "Cooling power: / %3.0f kW"; shows PLC_PRG.Oil_Water_Heat_Exchanger_Power.OIL_POWER
54 more shapes without text or variables
12 elements of other kinds (tables, trends, ...) not read
*)

(* Visualisation VISU_MENU
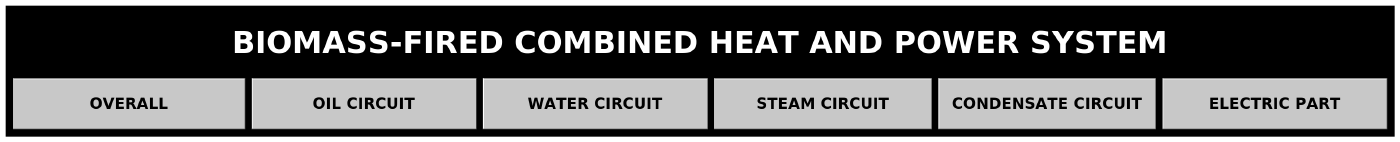
button at (10,100)-(331,171): text "OVERALL"; opens PLC_VISU
button at (340,100)-(651,171): text "OIL CIRCUIT"; opens PLC_VISU_OIL
button at (660,100)-(971,171): text "WATER CIRCUIT"; opens PLC_VISU_WATER
button at (980,100)-(1281,171): text "STEAM CIRCUIT"; opens PLC_VISU_STEAM
rectangle at (10,10)-(1911,91): text "BIOMASS-FIRED COMBINED HEAT AND POWER SYSTEM"
button at (1290,100)-(1591,171): text "CONDENSATE CIRCUIT"; opens PLC_VISU
button at (1600,100)-(1911,171): text "ELECTRIC PART"; opens PLC_VISU
1 more shapes without text or variables
*)
